# B&R Automation Studio project TD52 (part 137)

#### reactorCyclic.st
```iecst
 (*******************************************************************************
reactor		THERMOREACTOR

This code is confidential AND proprietary TO the INNIO Company.
It may NOT be used in any form, or reproduced in any manner,
without the express written permission OF the INNIO Company.
Copyright, INNIO Company, 2019

Customized modifications: -
------------------------

History:
-------
V15 	27-09-2001	Thaler, generated
V180	06-03-2003	Thaler, TR_ON_moduleTR, TR_OPER_moduleTR added. Connection to recipe REACTOR.
                            FGDRPS_moduleTR from FRG_GASREG_moduleTR --> reactor_a.
                            reactor_a --> TRW08.
V203	05-09-2003	Thaler, Modifications so that compatible with DIA.NE XT:
							y_HE_ramp INT --> UINT (reason: AS V2.3)
							Filter: 3 --> 10 (reason: AT664)
							DI_x: Value defined (reason: disabling #40 at Package Test).
							TK1, TK2 local --> global (reason: diagnosis for Development).
V210	28-09-2004	Thaler, TempInTR_moduleTR, TempOutTR_moduleTR, y_HE_Prom_moduleTR added.
							TK_GAS_OFF added.
							FG_HEIZG_moduleTR local --> global.
							TK_GAS.IN   := TK1_TK2_MIN; (war TK1_TK2_MIT).
							AN_PGW1 --> FG_TH_moduleTR.
V210.1	23-05-2006	Thaler, bExhReactor_moduleTR, Spuelluft-Ventil added.
V220    21-12-2007  Thaler, --> X20: variables declaration,
                            calculation Tvgl_moduleTR, iAT6402ETCreactor_moduleTR.
V220.2  27-05-2008  Thaler, DO_HE_xy added, TP_BTRB 180" --> DO_GAS_MINUS_moduleTR, ...
V250    12-03-2009  Thaler, UM_E_NEU_moduleTR: new position switches added.
                            TK_GAS_OFF settings changed.
V2.50.1 08-07-2009  Thaler, Spuelluft-Ventil modified.
                            Compensation_AI_TK_moduleTR added.
V3.20.0 11-03-2011  Thaler, with/without gas injection added:
                              sel_woGas: TK_w, TKx_y_HI_Gw, FRG_GASREG_moduleTR, PTON_KL_AUS
                              TK_w_woGas: TK_w
                              set_PT_KL_Pinc: PTON_KL_AUS
                              PT_KL_Pinc: PTON_KL_AUS.
                            alarm reset:
                              alarms unlatched for XT_Version_32x added
                              DI_QUITT_LT deleted (used for stand alone version only).
                            replaced variables:
                              M_GS_EIN --> DI_GCB_ON_moduleTR, NS_EIN -->  DI_MCB_ON_moduleTR
                            Spuelluft-Ventil modified:
                              TON_SPLU_AKT_AUS/EIN: 60s --> 10s
                              TON_SPLU_DEAKT: 60s --> 30s
V3.20.1 10-06-2011  Thaler, variabled deleted for simplifying Modular Software.
    	10-06-2011	Thaler, last modification
                            NOT compatible with other XT Versions !!

V04.00.00.00 	03-04-2014  Ganguly		HALio signals for 5 postion feedback and 4 postion feedback have same name,
							 			 in case of 4 position Mid-position feedback remains unconnected.
V04.03.00.00	25-09-2014	Denk		Bugfix, Flap switching time (INT/REAL casting)
										 Bugfix, KL_EIN renamed with OUT_TR.bThR_Val_SetIn
										 TRW01 : "FUEHLERBRUCH", TRW01_TempInOut and TRW01_Tvgl deleted
										 Bugfix, Sammelstoerung Reaktor Stop und Reaktor Stop + Motor Stop
V04.07.00.00	27-05-2019	Denk		Adjustments regarding new library versions (JEW_LIB1, JEW_LIB2, JEW_LIB3)
V04.09.00.00	09-03-2020	Denk		Bugfix, input variable changed in function xTON_TK1_DIF()
V04.12.00.00	19-05-2022	Maran		Bugfix: updated electrical heating elements switching logic and trigger signal for hour counter,
										 Bugfix: absolute value used for max. temperature difference detection in reactor vessel n.2,
										 Bugfix: HMI para used for aux.gas injection min. temperature hysteresis instead of fixed value,
										 removed unused TON for electrical heating thresholds detection
				14-06-2022	Maran		Removed unused TON for min.temperature detection to release auxiliary gas injection,
										 removed unused block of auxiliary gas injection release based on upper temperature bound
										 added A2356, A2357, A2358 in collective panel fault indication
V04.13.00.00	27-03-2023	Maran		Updated operating temperature definition and maximum temperature difference monitoring in TK1 and in TK2 (W3503)
				28-11-2023	Maran		Added W9374, W9375, W9376, W9377, W9381 in collective panel fault indication
V04.14.00.00	27-11-2024	Maran		Added auxiliary gas stop due to sufficient temperature,
										 temperature setpoint reference used in task changed from heating controller out structure value to HMI parameter value
				27-11-2024	Maran		Updates for thermal reactor 2nd generation (ThR2): revision of reactor chamber reference temperature,
										 added control of auxiliary gas solenoid valve before 4-way flap, adapted W3504 and blocked W3503,
										 added ThR2 chamber temperature signal fault to th.reactor bypass conditions, added ThR2 electrical heating control

Instructions for use:
--------------------

Outstandings:
------------
	FUB fuer ls und ls_t inkl. EN (ENABLE)
*******************************************************************************)
PROGRAM _CYCLIC

	xTON_INIT (IN:= TRUE, PT:= T#1m);
	OUT_TR.bThR_Active := xTON_INIT.Q AND IN_TR.tPB2MM.bParaSetupOk AND Para.bThR_Active;

	(* TK_moduleTR setpoint *)
	IF Para.bThR_woGas THEN
		TK_w := Para.rT_ThR_SetwoGas;    (* 0,1°C; without gas injection: see task "reac_set" *)
	ELSE
		TK_w := Para.tCtrTR_Heater.W_set;     (* Thermal reactor gas heating controller setpoint parameter *)
	END_IF;

	(* Temperature Limits [FB33] *)
	IF Para.bThR_woGas THEN
		TKx_y_HI_Gw       := 850.0;  (* 0,1°C; without gas injection: 850,0°C *)
	ELSE
		TKx_y_HI_Gw       := 800.0;  (* 0,1°C; with gas injection Standard: 800,0°C *)
	END_IF;

	(* Klappenumschaltzeit [FB40] *)
	(* Flap switching time *)
	PT_KL.x1 := REAL_TO_INT(TK_w + Para.rT_ThR_Val_x1);		(* von Rezept, 0,1°C; Standard: 20,0°C *)
	PT_KL.x2 := REAL_TO_INT(TK_w + Para.rT_ThR_Val_x2);		(* von Rezept, 0,1°C; Standard: 40,0°C *)
	PT_KL.y1 := TIME_TO_INT(Para.ti_ThR_Val_y1/1000);		(* von Rezept, Sekunden bei x1; Standard: 180s *)
	PT_KL.y2 := TIME_TO_INT(Para.ti_ThR_Val_y2/1000);		(* von Rezept, Sekunden bei x2; Standard: 360s *)

	(* Tvgl20_moduleTR von Rezept, 0,1°C; Standard: 0,0°C
	   Hier wird jener Wert angegeben,
	   den das Vergleichsstellenmessgeraet
	   bei 20° Umgebungstemperatur ausgibt. *)

	(******************************************************************************)
	(* Thermal Reactor temperature failure, min, max *)
	IF NOT Para.bThR2_Ena THEN //with Thermal reactor 1st generation
		MS_TK := (NOT IN_TR.tT_ThR_Chamber1_1.GoodQual) OR
				 (NOT IN_TR.tT_ThR_Chamber1_2.GoodQual) OR
				 (NOT IN_TR.tT_ThR_Chamber2_1.GoodQual) OR
				 (NOT IN_TR.tT_ThR_Chamber2_2.GoodQual);

		TK1 := (IN_TR.tT_ThR_Chamber1_1.Ai + IN_TR.tT_ThR_Chamber1_2.Ai)/2;
		TK2 := (IN_TR.tT_ThR_Chamber2_1.Ai + IN_TR.tT_ThR_Chamber2_2.Ai)/2;
	ELSE
		MS_TK := FALSE;
	END_IF
	IF Para.bThR2_Ena THEN //with Thermal reactor 2nd generation
		// individual measurement signal faults are defined with Thermal reactor 2, faults on left and right chamber are also used for reactor bypass
		bThR2_T_fault_ReactChamber := (NOT IN_TR.tThR2_T_UnitOk_RightCh.Di OR NOT IN_TR.tT_ThR2_RightChamber.GoodQual) OR
										(NOT IN_TR.tThR2_T_UnitOk_LeftCh.Di OR NOT IN_TR.tT_ThR2_LeftChamber.GoodQual);

		TK1 := IN_TR.tT_ThR2_RightChamber.Ai;
		TK2 := IN_TR.tT_ThR2_LeftChamber.Ai;
	ELSE
		bThR2_T_fault_ReactChamber := FALSE;
	END_IF

	TK1_TK2_MIT := (TK1 + TK2) / 2;
	TK1_TK2_MIN := MIN (TK1, TK2);
	TK1_TK2_MAX := MAX (TK1, TK2);
	(******************************************************************************)

	(* Steuerprogramm (aus PB4) *)

	(* Freigabe Thermoreaktor von Modulsteuerung *)
	(* Release Thermal Reactor from Module controller *)
	xTON_FG_TH (IN:= ((bThR_Rel AND IN_TR.tGCB_On.Di AND IN_TR.tMCB_On.Di) OR bThR_RelTest), PT:= T#30s);

	(* Freigabe Abgasklappen-Umschaltung und el. Heizung *)
	FG_KLUM						:= OUT_TR.bThR_Active AND xTON_FG_TH.Q AND
								    IN_TR.tThR_Swth_On.Di AND NOT ST_R_ST AND NOT ST_RM_ST;
	FG_HEIZG_moduleTR			:= FG_KLUM;
	OUT_TR.tThR_Contactor.Do	:= FG_HEIZG_moduleTR;
	OUT_TR.bThR_RelHeat			:= FG_HEIZG_moduleTR;

	(* Thermal Reactor auxiliary gas stop due to sufficient temperature *)
	bThr_AuxGasStopT_Ena := NOT Para.bThR_woGas AND Para.bThR_auxGasMonitor AND Para.bCtrThR_Heater_Active AND (TK_w > Para.rT_ThR_LimGas); (* check on parameters consistency *)

	xTON_Thr_AuxGasStopT_set(IN := OUT_TR.bThR_RelGas AND (IN_TR.tPos_ThR_AuxGasCV_Act.Ai < rPos_ThR_GasCV_AuxGasStop_max) (*CV essentially closed *) AND
	 IN_TR.tPos_ThR_AuxGasCV_Act.GoodQual AND (TK_moduleTR > TK_w + rT_Thr_AuxGasStopT_rel), PT := tiTON_Thr_AuxGasStopT_set);
	xRS_Thr_AuxGasStopT.SET := xTON_Thr_AuxGasStopT_set.Q; (* activation *)

	xTON_Thr_AuxGasStopT_reset(IN := (TK_moduleTR < TK_w), PT := tiTON_Thr_AuxGasStopT_reset);
	xRS_Thr_AuxGasStopT.RESET1 := xTON_Thr_AuxGasStopT_reset.Q OR NOT FG_HEIZG_moduleTR OR NOT bThr_AuxGasStopT_Ena; (* deactivation *)

	xRS_Thr_AuxGasStopT();

	(* Freigabe Einduesung *)
	OUT_TR.bThR_RelGas     := FG_HEIZG_moduleTR AND xTK_GAS.QH AND NOT Para.bThR_woGas AND NOT xRS_Thr_AuxGasStopT.Q1;
	OUT_TR.tThR_GT_COn1.Do := OUT_TR.bThR_RelGas;
	OUT_TR.tThR_GT_COn2.Do := OUT_TR.bThR_RelGas;
	OUT_TR.bThR_RelGas_Tmin	:= xTK_GAS.QH; (* minimum temperature for gas injection reached *)

	(* Betriebsmeldung *)
	OUT_TR.tThR_RunLamp.Do := (FG_KLUM AND (SEK_TAKT OR xTK_OPER.QH)) OR IN_TR.tThR_LampTest.Di;

	(* Betriebsmeldungen fuer auftragsbezogene Verwendung *)
	OUT_TR.bThR_Run         := FG_KLUM;               	    (* Reaktor eingeschaltet *)
	OUT_TR.bThR_RunReacTemp := FG_KLUM AND xTK_OPER.QH;	(* Reaktor eingeschaltet, Reaktionstemp. erreicht *)

	(* Ansteuerung Spuelluft-Stopp-Ventil, neu hinzu 07-2009 *)
	(* Aktivierung Spuelluft vor Durchfuehrung der Klappenbewegung *)
	PTON_SPLU_AKT_AUS := LIMIT (0, PTON_KL_AUS - T#10s, PTON_KL_AUS);
	PTON_SPLU_AKT_EIN := LIMIT (0, PTON_KL_EIN - T#10s, PTON_KL_EIN);
	xTON_SPLU_AKT_AUS (IN:= OUT_TR.bThR_Val_SetOut, PT:= PTON_SPLU_AKT_AUS);
	xTON_SPLU_AKT_EIN (IN:= OUT_TR.bThR_Val_SetIn, PT:= PTON_SPLU_AKT_EIN);

	(* Ansteuerung Spuelluft-Stopp-Ventil, neu hinzu 05-2006, modifiziert 07-2009 *)
	(* Deaktivierung Spuelluft nach Durchfuehrung der Klappenbewegung *)
	xTON_SPLU_DEAKT (IN:= (NOT FG_KLUM OR RM_KL_END), PT := T#30s);

	IF xTON_SPLU_DEAKT.Q THEN
		SPLU_AKT := FALSE;
	END_IF;

	(* IF FG_KLUM AND NOT OUT_TR.b_ThR_Val_SetIn AND NOT OUT_TR.b_ThR_Val_SetOut THEN *)
	IF (FG_KLUM AND NOT RM_KL_END) OR
	   (FG_KLUM AND (xTON_SPLU_AKT_AUS.Q OR xTON_SPLU_AKT_EIN.Q)) THEN
		SPLU_AKT := TRUE;
	END_IF;

	xTOF_W_INT (IN:= (IN_TR.tThR_Swth_On.Di AND xTON_W_ACT.Q), PT := T#10050m);	  (* weekly SPLU interval *)
	xTON_W_ACT (IN:= (IN_TR.tThR_Swth_On.Di AND NOT xTOF_W_INT.Q), PT := T#30m);  (* weekly SPLU active *)

	OUT_TR.tThR_Val_Air.Do := NOT (SPLU_AKT OR (IN_TR.tThR_Swth_On.Di AND NOT xTOF_W_INT.Q));	(* Ausgang fuer Spuelluft-Stopp-Ventil, TRUE bei STOP *)

	(* Klappensteuerung (aus OB13, FB35, FB36) *)

	(* Abgasklappe Mittelstellung: *)
	(* Im spannungslosen Zustand der Ansteuerventile geht die Klappe auf Mittelstellung. *)
	IF NOT FG_KLUM AND NOT Para.bSel_FlapActEl THEN
		OUT_TR.tThR_Val_CCylIn.Do  := FALSE;
		OUT_TR.tThR_Val_CCylOut.Do := FALSE;
	END_IF;

	(* Klappe Mittelstellung erreicht *)
	RM_KL_MIT :=          IN_TR.tPos_ThR_Val_Mid.Di
	              AND NOT IN_TR.tPos_ThR_Val_In1.Di
		          AND NOT IN_TR.tPos_ThR_Val_In2.Di
		          AND NOT IN_TR.tPos_ThR_Val_Out1.Di
				  AND NOT IN_TR.tPos_ThR_Val_Out2.Di;

	(* Abgasklappe Umschaltung: *)
	IF FG_KLUM THEN
		xR_TRIG_KL_AUS (CLK:= OUT_TR.bThR_Val_SetOut);
		xR_TRIG_KL_EIN (CLK:= OUT_TR.bThR_Val_SetIn);

		(* Bei positiver Flanke von KL_EIN_moduleTR oder KL_AUS_moduleTR sowie wenn KL_EIN_moduleTR und KL_AUS_moduleTR
		   nicht anstehen, wird die Mittelstellung aktiviert. *)
		IF (xR_TRIG_KL_AUS.Q OR xR_TRIG_KL_EIN.Q OR (OUT_TR.bThR_Val_SetOut AND OUT_TR.bThR_Val_SetIn)) THEN
			OUT_TR.tThR_Val_CCylIn.Do  := FALSE;
			OUT_TR.tThR_Val_CCylOut.Do := FALSE;
		END_IF;

		(* Klappe Ausfahren:
		   - Anfahren Mittelstellung durch Y1=0, Y2=0
		   - Rueckmeldung Mittelstellung erreicht: Ausfahren durch Aktivieren von Y2
		   - Ueberwachung:
		     Falls nach 10" die Endlage nicht erreicht wird,
		       "Stoerung Abgasklappe Ende" mit Reaktorabschaltung und
		       Befehl Abgasklappe Mittelstellung.
		     Falls 5" danach die Mittelstellung nicht erreicht wird,
		       "Stoerung Abgasklappe Mittelstellung" mit Gasmotorabstellung. *)
		IF OUT_TR.bThR_Val_SetOut THEN
			OUT_TR.tThR_Val_CCylIn.Do := FALSE;
		END_IF;

		IF (OUT_TR.bThR_Val_SetOut AND RM_KL_MIT) THEN
			OUT_TR.tThR_Val_CCylOut.Do := TRUE;
		END_IF;

		(* Klappe Einfahren:
		   - Anfahren Mittelstellung durch Y1=0, Y2=0
	   	   - Rueckmeldung Mittelstellung erreicht: Einfahren durch Aktivieren von Y1
		   - Ueberwachung:
		     Falls nach 10" die Endlage nicht erreicht wird,
		       "Stoerung Abgasklappe Ende" mit Reaktorabschaltung und
		       Befehl Abgasklappe Mittelstellung.
		     Falls 5" danach die Mittelstellung nicht erreicht wird,
		       "Stoerung Abgasklappe Mittelstellung" mit Gasmotorabstellung. *)
		IF OUT_TR.bThR_Val_SetIn THEN
			OUT_TR.tThR_Val_CCylOut.Do := FALSE;
		END_IF;

		IF (OUT_TR.bThR_Val_SetIn AND RM_KL_MIT) THEN
			OUT_TR.tThR_Val_CCylIn.Do := TRUE;
		END_IF;
	END_IF;

	(* Klappe Endlage erreicht *)
	RM_KL_END     := (	OUT_TR.bThR_Val_SetOut
					AND IN_TR.tPos_ThR_Val_Out1.Di
					AND IN_TR.tPos_ThR_Val_Out2.Di
					AND NOT IN_TR.tPos_ThR_Val_In1.Di
					AND NOT IN_TR.tPos_ThR_Val_In2.Di
					AND NOT IN_TR.tPos_ThR_Val_Mid.Di)
				  OR
					(	OUT_TR.bThR_Val_SetIn
					AND IN_TR.tPos_ThR_Val_In1.Di
					AND IN_TR.tPos_ThR_Val_In2.Di
					AND NOT IN_TR.tPos_ThR_Val_Out1.Di
					AND NOT IN_TR.tPos_ThR_Val_Out2.Di
					AND NOT IN_TR.tPos_ThR_Val_Mid.Di);

	RM_KL_END_AUS := (  IN_TR.tPos_ThR_Val_Out1.Di
					AND IN_TR.tPos_ThR_Val_Out2.Di
					AND NOT IN_TR.tPos_ThR_Val_In1.Di
					AND NOT IN_TR.tPos_ThR_Val_In2.Di
					AND NOT IN_TR.tPos_ThR_Val_Mid.Di);

	RM_KL_END_EIN := (  IN_TR.tPos_ThR_Val_In1.Di
					AND IN_TR.tPos_ThR_Val_In2.Di
					AND NOT IN_TR.tPos_ThR_Val_Out1.Di
					AND NOT IN_TR.tPos_ThR_Val_Out2.Di
					AND NOT IN_TR.tPos_ThR_Val_Mid.Di);

	(* Abgasklappe Einschaltung Schütze mit E-Antrieb: *)
	(* Abgasklappe Mittelstellung mit E-Antrieb: *)
	IF NOT FG_KLUM AND Para.bSel_FlapActEl THEN
		R_TRIG_KL_AUS_M (CLK:= KL_AUS_M);
		R_TRIG_KL_EIN_M (CLK:= KL_EIN_M);
		OUT_TR.tThR_Val_CCylOut.Do := R_TRIG_KL_AUS_M.Q;
		OUT_TR.tThR_Val_CCylIn.Do  := R_TRIG_KL_EIN_M.Q;
	END_IF;
	(* Anmerkung: Selbsthaltung extern mit Schütz, Absteuerung mit Endschalter Mittelstellung *)

	(* Abgasklappe Umschaltung mit E-Antrieb: *)
	IF FG_KLUM AND Para.bSel_FlapActEl THEN

		(* Klappe Ausfahren:
	   	   - Rueckmeldung Endlage_Eingefahren oder Mittelstellung erreicht:
	         Ausfahren durch Dauerbefehl *)

		(* Dauerbefehl fuer Richtungswechsel *)
		IF (OUT_TR.bThR_Val_SetOut AND (RM_KL_MIT OR RM_KL_END_EIN)) THEN
			OUT_TR.tThR_Val_CCylOut.Do := TRUE;
		END_IF;

		(* Klappe Einfahren:
	   	   - Rueckmeldung Endlage_Ausgefahren oder Mittelstellung erreicht:
	         Einfahren durch Dauerbefehl *)

		(* Dauerbefehl fuer Richtungswechsel *)
		IF (OUT_TR.bThR_Val_SetIn AND (RM_KL_MIT OR RM_KL_END_AUS)) THEN
			OUT_TR.tThR_Val_CCylIn.Do := TRUE;
		END_IF;
	END_IF;

	(* Zeittakte Abgasklappe Umschaltung *)
	OUT_TR.bThR_Val_SetOut  := FG_KLUM
							AND (NOT xTON_KL_AUS.Q)
							AND (NOT OUT_TR.bThR_Val_SetIn)
							AND (OUT_TR.bThR_Val_SetOut OR NOT KL_AUS_S);

	IF OUT_TR.bThR_Val_SetOut THEN
		KL_AUS_S   := TRUE;
		KL_AUS_M_S := TRUE;
		KL_EIN_S   := FALSE;
		KL_EIN_M_S := FALSE;
	END_IF;
	xTON_KL_AUS (IN:= OUT_TR.bThR_Val_SetOut, PT:= PTON_KL_AUS);

	OUT_TR.bThR_Val_SetIn := FG_KLUM
						AND (NOT xTON_KL_EIN.Q)
						AND (NOT OUT_TR.bThR_Val_SetOut)
						AND TRUE;

	IF OUT_TR.bThR_Val_SetIn THEN
		KL_EIN_S   := TRUE;
		KL_EIN_M_S := TRUE;
		KL_AUS_S   := FALSE;
		KL_AUS_M_S := FALSE;
	END_IF;
	xTON_KL_EIN (IN:= OUT_TR.bThR_Val_SetIn, PT:= PTON_KL_EIN);

	(* Abgasklappe Mittelstellung mit E-Antrieb: *)
	(* Zeittakte Abgasklappe für Anfahren Mittelstellung mit E-Antrieb: *)
	xTOF_S_EIN (IN:= (Para.bThR_Active AND IN_TR.tThR_Swth_On.Di), PT:= T#15s);
	xTON_FG_KL_M (IN:= (xTOF_S_EIN.Q AND NOT FG_KLUM AND NOT RM_KL_MIT AND NOT xTRA01M.Q1), PT:= T#1s);
	FG_KL_M := xTON_FG_KL_M.Q;

	KL_AUS_M := FG_KL_M AND NOT xTON_KL_AUS_M.Q AND NOT KL_EIN_M AND
				(KL_AUS_M OR NOT KL_AUS_M_S OR RM_KL_END_EIN);
	IF KL_AUS_M THEN
		KL_AUS_M_S := TRUE;
		KL_EIN_M_S := FALSE;
	END_IF;
	xTON_KL_AUS_M (IN:= KL_AUS_M, PT:= T#5s);

	KL_EIN_M := FG_KL_M AND NOT xTON_KL_EIN_M.Q AND NOT KL_AUS_M AND TRUE;
	IF KL_EIN_M THEN
		KL_EIN_M_S := TRUE;
		KL_AUS_M_S := FALSE;
	END_IF;
	xTON_KL_EIN_M (IN:= KL_EIN_M, PT:= T#5s);

	(* Abgasklappe Umschaltung mit E-Antrieb: *)
	IF FG_KLUM AND Para.bSel_FlapActEl THEN

		(* Klappe Ausfahren:
	       - Rueckmeldung Endlage_Eingefahren oder Mittelstellung erreicht:
	         Ausfahren durch Dauerbefehl (siehe oberhalb)
	       - Rueckmeldung Endlage_Ausgefahren: Beendigung Dauerbefehl
	       - Ueberwachung:
	         Falls nach 10" die Endlage nicht erreicht wird,
	         "Stoerung Abgasklappe Ende" mit Reaktorabschaltung und
	         Befehl Abgasklappe Mittelstellung.
	         Falls 5" danach die Mittelstellung nicht erreicht wird,
	         "Stoerung Abgasklappe Mittelstellung" mit Gasmotorabstellung. *)

		(* Absteuerung *)
		IF (OUT_TR.bThR_Val_SetOut AND RM_KL_END_AUS) OR NOT OUT_TR.bThR_Val_SetOut THEN
			OUT_TR.tThR_Val_CCylOut.Do := FALSE;
		END_IF;

		(* Klappe Einfahren:
	   	   - Rueckmeldung Endlage_Ausgefahren oder Mittelstellung erreicht:
	      	 Einfahren durch Dauerbefehl (siehe oberhalb)
	   	   - Rueckmeldung Endlage_Eingefahren: Beendigung Dauerbefehl
	   	   - Ueberwachung:
	     	 Falls nach 10" die Endlage nicht erreicht wird,
	       	 "Stoerung Abgasklappe Ende" mit Reaktorabschaltung und
	       	 Befehl Abgasklappe Mittelstellung.
	     	 Falls 5" danach die Mittelstellung nicht erreicht wird,
	       	 "Stoerung Abgasklappe Mittelstellung" mit Gasmotorabstellung. *)

		(* Absteuerung *)
		IF (OUT_TR.bThR_Val_SetIn AND RM_KL_END_EIN) OR NOT OUT_TR.bThR_Val_SetIn THEN
			OUT_TR.tThR_Val_CCylIn.Do  := FALSE;
		END_IF;
	END_IF;

	(* Abgasklappe Verriegelung mit E-Antrieb: *)
	IF Para.bSel_FlapActEl THEN
		IF OUT_TR.bThR_Val_SetOut OR KL_AUS_M THEN
			OUT_TR.tThR_Val_CCylIn.Do  := FALSE;
		END_IF;
		IF OUT_TR.bThR_Val_SetIn OR KL_EIN_M THEN
			OUT_TR.tThR_Val_CCylOut.Do  := FALSE;
		END_IF;
	END_IF;

	(* Abgasklappe Mittelstellung mit Druckluft-Anztrieb: *)
	(* Im spannungslosen Zustand der Ansteuerventile geht die Klappe auf Mittelstellung. *)
	IF NOT FG_KLUM AND NOT Para.bSel_FlapActEl THEN
		OUT_TR.tThR_Val_CCylIn.Do  := FALSE;
		OUT_TR.tThR_Val_CCylOut.Do := FALSE;
	END_IF;

	(* Abgasklappe Umschaltung mit Druckluft-Antrieb: *)
	IF FG_KLUM AND NOT Para.bSel_FlapActEl THEN
		R_TRIG_KL_AUS (CLK:= OUT_TR.bThR_Val_SetOut);
		R_TRIG_KL_EIN (CLK:= OUT_TR.bThR_Val_SetIn);

		(* Bei positiver Flanke von KL_EIN oder KL_AUS sowie wenn KL_EIN und KL_AUS
	    nicht anstehen, wird die Mittelstellung aktiviert. *)
		IF (R_TRIG_KL_AUS.Q OR R_TRIG_KL_EIN.Q OR (OUT_TR.bThR_Val_SetOut AND OUT_TR.bThR_Val_SetIn)) THEN
			OUT_TR.tThR_Val_CCylIn.Do  := FALSE;
			OUT_TR.tThR_Val_CCylOut.Do := FALSE;
		END_IF;

		(* Klappe Ausfahren:
	       - Anfahren Mittelstellung durch Y1=0, Y2=0
	       - Rueckmeldung Mittelstellung erreicht: Ausfahren durch Aktivieren von Y2
	       - Ueberwachung:
	       Falls nach 10" die Endlage nicht erreicht wird,
	       "Stoerung Abgasklappe Ende" mit Reaktorabschaltung und
	       Befehl Abgasklappe Mittelstellung.
	       Falls 5" danach die Mittelstellung nicht erreicht wird,
	       "Stoerung Abgasklappe Mittelstellung" mit Gasmotorabstellung. *)
		IF OUT_TR.bThR_Val_SetOut THEN
			OUT_TR.tThR_Val_CCylIn.Do := FALSE;
		END_IF;
		IF (OUT_TR.bThR_Val_SetOut AND RM_KL_MIT) THEN
			OUT_TR.tThR_Val_CCylOut.Do := TRUE;
		END_IF;

		(* Klappe Einfahren:
	   	   - Anfahren Mittelstellung durch Y1=0, Y2=0
	  	   - Rueckmeldung Mittelstellung erreicht: Einfahren durch Aktivieren von Y1
	       - Ueberwachung:
	     		Falls nach 10" die Endlage nicht erreicht wird,
	       		"Stoerung Abgasklappe Ende" mit Reaktorabschaltung und
	            Befehl Abgasklappe Mittelstellung.
	     		Falls 5" danach die Mittelstellung nicht erreicht wird,
	       		"Stoerung Abgasklappe Mittelstellung" mit Gasmotorabstellung. *)
		IF OUT_TR.bThR_Val_SetIn THEN
			OUT_TR.tThR_Val_CCylOut.Do := FALSE;
		END_IF;
		IF (OUT_TR.bThR_Val_SetIn AND RM_KL_MIT) THEN
			OUT_TR.tThR_Val_CCylIn.Do := TRUE;
		END_IF;
	END_IF;

	(* Thermal Reactor auxiliary gas solenoid valve - ThR2 *)
	IF Para.bThR2_Ena THEN
		IF OUT_TR.bThR_RelGas THEN
			//update blockage function inputs before 4-way flap switching request depending on last end-position
			IF iThr2_lastFlapEndPosIndex = 1 THEN
				xSR_Thr2_AuxGasValve_Block.SET1 := xTON_KL_EIN.PT - xTON_KL_EIN.ET <= tiThR2_AuxGasValve_Block;
				xSR_Thr2_AuxGasValve_Block.RESET := RM_KL_END_AUS;
			ELSIF iThr2_lastFlapEndPosIndex = -1 THEN
				xSR_Thr2_AuxGasValve_Block.SET1 := xTON_KL_AUS.PT - xTON_KL_AUS.ET <= tiThR2_AuxGasValve_Block;
				xSR_Thr2_AuxGasValve_Block.RESET := RM_KL_END_EIN;
			END_IF
		ELSE //reinitialize blockage function inputs in case of Th.Reactor aux.gas system stop
			xSR_Thr2_AuxGasValve_Block.SET1 := FALSE;
			xSR_Thr2_AuxGasValve_Block.RESET := TRUE;
		END_IF
		xSR_Thr2_AuxGasValve_Block();
		OUT_TR.tThR2_AuxGasShutOffValve_Dem.Do := OUT_TR.bThR_RelGas AND RM_KL_END AND (NOT xSR_Thr2_AuxGasValve_Block.Q1);
	ELSE
		//reset SR in IF block
		xSR_Thr2_AuxGasValve_Block.SET1 := FALSE;
		xSR_Thr2_AuxGasValve_Block.RESET := TRUE;
		//reset output signal gas solenoid valve - ThR2
		OUT_TR.tThR2_AuxGasShutOffValve_Dem.Do := FALSE;
	END_IF
	IF OUT_TR.bThR_RelGas THEN //record last end-position reached by 4-way flap during aux. gas. injection operation
		IF RM_KL_END_EIN THEN
			iThr2_lastFlapEndPosIndex := 1; //right position
		ELSIF RM_KL_END_AUS THEN
			iThr2_lastFlapEndPosIndex := -1; //left position
		END_IF
	ELSE
		iThr2_lastFlapEndPosIndex := 0; //reset position index
	END_IF

	//block the auxiliary gas heating controller if corresponding solenoid valve is closed
	bThr2_AuxGasValve_CtrlBlock := Para.bThR2_Ena AND OUT_TR.bThR_RelGas AND NOT OUT_TR.tThR2_AuxGasShutOffValve_Dem.Do;

	(******************************************************************************)
	(******************************************************************************)

	(* Ueberwachungen [PB45] *)

	(* TRA01 : "STOERUNG ABGASKLAPPE MITTELSTELLUNG" *)
	xTON_ST_KLM.IN := OUT_TR.bThR_Active AND NOT FG_KLUM AND NOT RM_KL_MIT AND NOT xTON_ST_KLM.Q AND NOT xTRA01M.RESET;
	xTON_ST_KLM.PT := T#15s;
	xTON_ST_KLM;
	xTRA01.SET1  := xTON_ST_KLM.Q;
	xTRA01.RESET := NOT xTRA01.SET1;
	xTRA01();
	xTRA01M.SET1  := xTON_ST_KLM.Q;
	xTRA01M.RESET := IN_TR.tAB2TR.bResetTrip;
	xTRA01M();

	(* TRA02 : "SICHERHEITSSCHLEIFE THERMOREAKTOR", aktiv nur bei RIO *)
	xTRA02.SET1  := IN_TR.tThR_SL.Di;
	xTRA02.RESET := NOT xTRA02.SET1;
	xTRA02();

	(* TRW01 : "FUEHLERBRUCH" *)
	xTRW01_TK.SET1  := MS_TK;
	xTRW01_TK.RESET := NOT xTRW01_TK.SET1;
	xTRW01_TK();
	xTRW01.SET1  := xTRW01_TK.Q1;
	xTRW01.RESET := NOT xTRW01.SET1;
	xTRW01();

	(* TRW02 : "STOERUNG DRUCKLUFTVERSORGUNG" *)
	xTOF_PS_LUFT (IN:= IN_TR.tPr_ThR_AirLo.Di  AND NOT Para.bSel_FlapActEl, PT := T#10s);
	xTRW02.SET1  := Para.bThR_Active AND NOT xTOF_PS_LUFT.Q AND NOT Para.bSel_FlapActEl;
	xTRW02.RESET := NOT xTRW02.SET1;
	xTRW02();

	(* TRW03 : "STOERUNG ABGASKLAPPE ENDLAGE" *)
	xTON_ST_KLE (IN:= ((OUT_TR.bThR_Val_SetOut AND NOT RM_KL_END_AUS) OR
					   (OUT_TR.bThR_Val_SetIn  AND NOT RM_KL_END_EIN)), PT:= T#10s);
	xTRW03.SET1  := xTON_ST_KLE.Q;
	xTRW03.RESET := NOT xTRW03.SET1;
	xTRW03();

	(* TRW04 : "AUFHEIZZEIT UEBERSCHRITTEN" *)
	xTON_AUFHEIZG_GES (IN:= (FG_KLUM AND NOT xTK_OPER.QH), PT:= T#600m);
	xTON_AUFHEIZG_GAS (IN:= (OUT_TR.bThR_RelGas AND NOT xTK_OPER.QH), PT:= T#300m);
	xTRW04.SET1  := xTON_AUFHEIZG_GES.Q OR xTON_AUFHEIZG_GAS.Q;
	xTRW04.RESET := NOT xTRW04.SET1;
	xTRW04();

	(* TRW05 : "SCHALTSCHRANKTEMPERATUR MAXIMUM" *)
	xTRW05.SET1  := OUT_TR.bThR_Active AND NOT IN_TR.tT_ThR_Swg_Hi.Di;
	xTRW05.RESET := NOT xTRW05.SET1;
	xTRW05();

	(* TRW06 : "ZULAESSIGE DIFFERENZ VON TEMPERATUREN TK1/TK2 UEBER MAXIMUM" *)
	xTRW06.SET1  := xTK1_DIF_HI.QH OR xTK2_DIF_HI.QH;
	xTRW06.RESET := NOT xTRW06.SET1;
	xTRW06();

	(* TRW07 : "TEMPERATUR REAKTIONSKAMMER TK1/TK2 MAXIMUM" *)
	IF NOT Para.bThR2_Ena THEN //with Thermal reactor 1st generation
		xTRW07.SET1  := xTK1_1_HI.QH OR xTK1_2_HI.QH OR xTK2_1_HI.QH OR xTK2_2_HI.QH;
	END_IF
	IF Para.bThR2_Ena THEN //with Thermal reactor 2nd generation
	   (*************** temperature threshold check for TRW07 - ThR2 ***************)
		xGRMax_ThR2_T_LeftChamber_Hi(Gw := TKx_y_HI_Gw, Hy := TKx_y_HI_Hy, In := IN_TR.tT_ThR2_LeftChamber.Ai);
		xTON_ThR2_T_LeftChamber_Hi(IN := xGRMax_ThR2_T_LeftChamber_Hi.Q, PT := ti_TKx_y_HI_PTHI);

		xGRMax_ThR2_T_RightChamber_Hi(Gw := TKx_y_HI_Gw, Hy := TKx_y_HI_Hy, In := IN_TR.tT_ThR2_RightChamber.Ai);
		xTON_ThR2_T_RightChamber_Hi(IN := xGRMax_ThR2_T_RightChamber_Hi.Q, PT := ti_TKx_y_HI_PTHI);

		xTRW07.SET1  := xTON_ThR2_T_LeftChamber_Hi.Q OR xTON_ThR2_T_RightChamber_Hi.Q;
	ELSE //reset TON in IF block
		xTON_ThR2_T_LeftChamber_Hi(IN := FALSE, PT := ti_TKx_y_HI_PTHI);
		xTON_ThR2_T_RightChamber_Hi(IN := FALSE, PT := ti_TKx_y_HI_PTHI);
	END_IF
	xTRW07.RESET := NOT xTRW07.SET1;
	xTRW07();

	(* TRW08 : "TEMPERATUR REAKTIONSKAMMER MINIMUM" *)
	xTRW08.SET1  := OUT_TR.bThR_Active AND NOT IN_TR.tT_ThR_ChamberLo.Di;
	xTRW08.RESET := NOT xTRW08.SET1;
	xTRW08();

	(* Sammelstoerung Reaktor Stop *)
	IF IN_TR.tAB2TR.bResetWarning THEN
		ST_R_ST := FALSE;
	END_IF;

	IF (xTRW01_TK.Q1
		OR bThR2_T_fault_ReactChamber
		OR xTRW02.Q1
		OR xTRW03.Q1
		OR xTRW04.Q1
		OR xTRW05.Q1
		OR xTRW06.Q1
		OR xTRW07.Q1
		OR xTRW08.Q1) THEN
		ST_R_ST := TRUE;
	END_IF;

	(* Sammelstoerung Reaktor + Motor Stop *)
	IF IN_TR.tAB2TR.bResetTrip THEN
		ST_RM_ST := FALSE;
	END_IF;

	IF FALSE (* priority 3 alarms from Th.Reactor to be included here *) THEN
		 ST_RM_ST := TRUE;
	END_IF;

	(* H2: "Reaktor Sammelstoerung", aktiv nur bei RIO *)
	OUT_TR.tThR_ErrLamp.Do
		:= xTRA01.Q1
		OR xTRA02.Q1
		OR MM2VIS.bMsg2356
		OR MM2VIS.bMsg2357
		OR MM2VIS.bMsg2358
		OR xTRW01.Q1
		OR bThR2_T_fault_ReactChamber
		OR xTRW02.Q1
		OR xTRW03.Q1
		OR xTRW04.Q1
		OR xTRW05.Q1
		OR xTRW06.Q1
		OR xTRW07.Q1
		OR xTRW08.Q1
		OR MM2VIS.bMsg9374
		OR MM2VIS.bMsg9375
		OR MM2VIS.bMsg9376
		OR MM2VIS.bMsg9377
		OR MM2VIS.bMsg9381
		OR IN_TR.tThR_LampTest.Di;

	(******************************************************************************)
	(* Auswahl der Reaktionstemperatur in Abhaengigkeit der Stroemungsrichtung [FB66] *)
	TK_moduleTR := TK1_TK2_MAX;

	(* Sekundentakt [FB3]
	CTU_SEK_TAKT (CU := FALSE, RESET := CTU_SEK_TAKT.Q, PV := 10);
	CTU_SEK_TAKT (CU := TRUE, RESET := CTU_SEK_TAKT.Q, PV := 10);
	SEK_TAKT := (CTU_SEK_TAKT.CV >= 5) AND (CTU_SEK_TAKT.CV <= 10);
	*)

	xTON_reactor_01.IN := NOT(SEK_TAKT);
	xTON_reactor_01.PT := T#300ms;
	xTON_reactor_01();

	IF (xTON_reactor_01.Q = 1) THEN
		SEK_TAKT := 1;
	END_IF;

	xTON_reactor_02.IN := SEK_TAKT;
	xTON_reactor_02.PT := T#600ms;
	xTON_reactor_02();

	IF (xTON_reactor_02.Q = 1) THEN
		SEK_TAKT := 0;
	END_IF;

	IF NOT Para.bThR2_Ena THEN // El. heating with Thermal reactor 1st generation
		(* Heizstabsteuerung [FB45, FB56]
		   Periodendauer = 4*100ms.
		   Impulsdauer   = 0...4*100ms. *)
		xCTD_HE_1 (CD := FALSE, LOAD := xCTD_HE_1.Q, PV := 4);
		xCTD_HE_1 (CD := TRUE, LOAD := xCTD_HE_1.Q, PV := 4);

		(* Phasenverschiebung 2*100ms *)
		xCTD_HE_2 (CD := FALSE, LOAD := xCTD_HE_1.CV = 1, PV := 4);
		xCTD_HE_2 (CD := TRUE, LOAD := FALSE, PV := 4);

		(* Phasenverschiebung 3*100ms *)
		xCTD_HE_3 (CD := FALSE, LOAD := xCTD_HE_1.CV = 0, PV := 4);
		xCTD_HE_3 (CD := TRUE, LOAD := FALSE, PV := 4);

		IF FG_HEIZG_moduleTR = FALSE OR xTK_E00.QH THEN
			y_HE := 0;
		ELSIF FG_HEIZG_moduleTR AND NOT(xTK_E00.QH) AND xTK_E25.QH THEN
			y_HE := 1;
		ELSIF FG_HEIZG_moduleTR AND NOT(xTK_E00.QH) AND NOT(xTK_E25.QH) AND xTK_E50.QH THEN
			y_HE := 2;
		ELSIF FG_HEIZG_moduleTR AND NOT(xTK_E00.QH) AND NOT(xTK_E25.QH) AND NOT(xTK_E50.QH) AND xTK_E75.QH THEN
			y_HE := 3;
		ELSIF FG_HEIZG_moduleTR AND NOT(xTK_E00.QH) AND NOT(xTK_E25.QH) AND NOT(xTK_E50.QH) AND NOT(xTK_E75.QH) THEN
			y_HE := 4;
		ELSE
			y_HE := 0;
		END_IF;

		(* RAMP FUNCTION *)
		P_ramp[0].In         := REAL_TO_INT(y_HE * 1000);      (* "PV_In": use "PV Name" of "In" *)
		P_ramp[0].In_ref     := 1;                (* reference value, units like "In" *)
		P_ramp[0].mode       := 0;                (* 1: dOut=Ki*(In-Out)/In_ref, 0: dOut=Ki *)
		P_ramp[0].Ki_plus    := 333;              (* 0,1 units "In"/s *)
		P_ramp[0].Ki_minus   := 10000;            (* 0,1 units "In"/s *)
		P_ramp[0].dOut_max_p := 10000;            (* 0,1 units "In"/s *)
		P_ramp[0].dOut_max_m := 10000;            (* 0,1 units "In"/s *)
		P_ramp[0].Out_min    := 0;                (* units like "In" *)
		P_ramp[0].Out_max    := P_ramp[0].In;     (* units like "In" *)
		y_HE_ramp := REAL_TO_UINT(P_ramp[0].Out) / 1000;	(* "PV_Out": use "PV Name" of "Out", units like "In" *)

		rThR_EH_pulse := LIMIT(0, UINT_TO_REAL(y_HE_ramp * 100) - 10, 290);	// limit pulse duration from 0% to 75% of time interval
		tThR_EH_pulse:= REAL_TO_TIME(rThR_EH_pulse);
		xTP_EH11(IN := xCTD_HE_1.Q, PT:= tThR_EH_pulse);
		xTP_EH21(IN := xCTD_HE_2.Q, PT:= tThR_EH_pulse);
		xTP_EH31(IN := xCTD_HE_3.Q, PT:= tThR_EH_pulse);
		OUT_TR.tThR_EH11.Do := xTP_EH11.Q;
		OUT_TR.tThR_EH21.Do := xTP_EH21.Q;
		OUT_TR.tThR_EH31.Do := xTP_EH31.Q;
		IF y_HE_ramp = 4 THEN 												// overwrite pulse signal for 100% heating output request
			OUT_TR.tThR_EH11.Do := OUT_TR.tThR_EH21.Do := OUT_TR.tThR_EH31.Do := 1;
		END_IF
		IF y_HE_ramp = 0 THEN 												// overwrite pulse signal for no heating output request
			OUT_TR.tThR_EH11.Do := OUT_TR.tThR_EH21.Do := OUT_TR.tThR_EH31.Do := 0;
		END_IF

		OUT_TR.tThR_EH12.Do := OUT_TR.tThR_EH11.Do;
		OUT_TR.tThR_EH13.Do := OUT_TR.tThR_EH11.Do;

		OUT_TR.tThR_EH22.Do := OUT_TR.tThR_EH21.Do;
		OUT_TR.tThR_EH23.Do := OUT_TR.tThR_EH21.Do;

		OUT_TR.tThR_EH32.Do := OUT_TR.tThR_EH31.Do;
		OUT_TR.tThR_EH33.Do := OUT_TR.tThR_EH31.Do;

		IF FG_HEIZG_moduleTR THEN
			CASE y_HE_ramp OF
				0: OUT_TR.rP_ThR_EH := 0;
				1: OUT_TR.rP_ThR_EH := 250;
				2: OUT_TR.rP_ThR_EH := 500;
				3: OUT_TR.rP_ThR_EH := 750;
				4: OUT_TR.rP_ThR_EH := 1000;
			ELSE
				OUT_TR.rP_ThR_EH := 0;
			END_CASE;
		ELSE
			OUT_TR.rP_ThR_EH := 0;
		END_IF;

	ELSE
		//reset ramps/timer blocks in IF block
		P_ramp[0].Out_internal := 0;
		P_ramp[1].Out_internal := 0; //P_ramp[1] never used, reinitialized for completeness
		xTP_EH11(IN := FALSE);
		xTP_EH21(IN := FALSE);
		xTP_EH31(IN := FALSE);
	END_IF
	IF Para.bThR2_Ena THEN // El. heating with Thermal reactor 2nd generation
		//definition of five el.heating power levels
		xGRMax_ThR2_EH_pw00(Gw := Para.rT_ThR2_EH_Lim00, Hy := rT_ThR2_EH_PwLevHy, In := TK_moduleTR);
		xGRMax_ThR2_EH_pw20(Gw := Para.rT_ThR2_EH_Lim20, Hy := rT_ThR2_EH_PwLevHy, In := TK_moduleTR);
		xGRMax_ThR2_EH_pw40(Gw := Para.rT_ThR2_EH_Lim40, Hy := rT_ThR2_EH_PwLevHy, In := TK_moduleTR);
		xGRMax_ThR2_EH_pw60(Gw := Para.rT_ThR2_EH_Lim60, Hy := rT_ThR2_EH_PwLevHy, In := TK_moduleTR);
		xGRMax_ThR2_EH_pw80(Gw := Para.rT_ThR2_EH_Lim80, Hy := rT_ThR2_EH_PwLevHy, In := TK_moduleTR);

		IF FG_HEIZG_moduleTR = FALSE OR xGRMax_ThR2_EH_pw00.Q THEN
			iThR2_EH_PwLev := 0;
		ELSIF FG_HEIZG_moduleTR AND NOT(xGRMax_ThR2_EH_pw00.Q) AND xGRMax_ThR2_EH_pw20.Q THEN
			iThR2_EH_PwLev := 1;
		ELSIF FG_HEIZG_moduleTR AND NOT(xGRMax_ThR2_EH_pw00.Q) AND NOT(xGRMax_ThR2_EH_pw20.Q) AND xGRMax_ThR2_EH_pw40.Q THEN
			iThR2_EH_PwLev := 2;
		ELSIF FG_HEIZG_moduleTR AND NOT(xGRMax_ThR2_EH_pw00.Q) AND NOT(xGRMax_ThR2_EH_pw20.Q) AND NOT(xGRMax_ThR2_EH_pw40.Q) AND xGRMax_ThR2_EH_pw60.Q THEN
			iThR2_EH_PwLev := 3;
		ELSIF FG_HEIZG_moduleTR AND NOT(xGRMax_ThR2_EH_pw00.Q) AND NOT(xGRMax_ThR2_EH_pw20.Q) AND NOT(xGRMax_ThR2_EH_pw40.Q) AND NOT(xGRMax_ThR2_EH_pw60.Q) AND xGRMax_ThR2_EH_pw80.Q THEN
			iThR2_EH_PwLev := 4;
		ELSIF FG_HEIZG_moduleTR AND NOT(xGRMax_ThR2_EH_pw00.Q) AND NOT(xGRMax_ThR2_EH_pw20.Q) AND NOT(xGRMax_ThR2_EH_pw40.Q) AND NOT(xGRMax_ThR2_EH_pw60.Q) AND NOT(xGRMax_ThR2_EH_pw80.Q) THEN
			iThR2_EH_PwLev := 5;
		ELSE
			iThR2_EH_PwLev := 0;
		END_IF;

		//time ramp for el.heating power level
		xRamp_ThR2_EH_PwLev.In := INT_TO_REAL(iThR2_EH_PwLev);
		xRamp_ThR2_EH_PwLev();
		iThR2_EH_PwLev_ramp := TRUNC(xRamp_ThR2_EH_PwLev.Out);
		OUT_TR.rP_ThR_EH := INT_TO_REAL(iThR2_EH_PwLev_ramp) / 5 * 1000; (* 5 el.heating power levels, 1000 HMI display scaling factor *)

		//monitoring of heating elements groups availability depending on max.temperature
		xTON_ThR2_EH_gr1_T_GoodQual(IN := IN_TR.tT_ThR2_EH_group1.GoodQual, PT := tiTON_ThR2_EH_gr_T_GoodQual);
		xTON_ThR2_EH_gr2_T_GoodQual(IN := IN_TR.tT_ThR2_EH_group2.GoodQual, PT := tiTON_ThR2_EH_gr_T_GoodQual);
		xTON_ThR2_EH_gr3_T_GoodQual(IN := IN_TR.tT_ThR2_EH_group3.GoodQual, PT := tiTON_ThR2_EH_gr_T_GoodQual);
		xTON_ThR2_EH_gr4_T_GoodQual(IN := IN_TR.tT_ThR2_EH_group4.GoodQual, PT := tiTON_ThR2_EH_gr_T_GoodQual);
		xTON_ThR2_EH_gr5_T_GoodQual(IN := IN_TR.tT_ThR2_EH_group5.GoodQual, PT := tiTON_ThR2_EH_gr_T_GoodQual);

		xGRMax_ThR2_EH_group1_T(Gw := rT_ThR2_EH_thres_GroupHi, Hy := rT_ThR2_EH_thres_GroupHi_Hy, In := IN_TR.tT_ThR2_EH_group1.Ai);
		bThR2_EH_gr1_T_blocked := xGRMax_ThR2_EH_group1_T.Q AND xTON_ThR2_EH_gr1_T_GoodQual.Q;
		bThR2_EH_groupT_Ok[1] := NOT bThR2_EH_gr1_T_blocked;
		xGRMax_ThR2_EH_group2_T(Gw := rT_ThR2_EH_thres_GroupHi, Hy := rT_ThR2_EH_thres_GroupHi_Hy, In := IN_TR.tT_ThR2_EH_group2.Ai);
		bThR2_EH_gr2_T_blocked := xGRMax_ThR2_EH_group2_T.Q AND xTON_ThR2_EH_gr2_T_GoodQual.Q;
		bThR2_EH_groupT_Ok[2] := NOT bThR2_EH_gr2_T_blocked;
		xGRMax_ThR2_EH_group3_T(Gw := rT_ThR2_EH_thres_GroupHi, Hy := rT_ThR2_EH_thres_GroupHi_Hy, In := IN_TR.tT_ThR2_EH_group3.Ai);
		bThR2_EH_gr3_T_blocked := xGRMax_ThR2_EH_group3_T.Q AND xTON_ThR2_EH_gr3_T_GoodQual.Q;
		bThR2_EH_groupT_Ok[3] := NOT bThR2_EH_gr3_T_blocked;
		xGRMax_ThR2_EH_group4_T(Gw := rT_ThR2_EH_thres_GroupHi, Hy := rT_ThR2_EH_thres_GroupHi_Hy, In := IN_TR.tT_ThR2_EH_group4.Ai);
		bThR2_EH_gr4_T_blocked := xGRMax_ThR2_EH_group4_T.Q AND xTON_ThR2_EH_gr4_T_GoodQual.Q;
		bThR2_EH_groupT_Ok[4] := NOT bThR2_EH_gr4_T_blocked;
		xGRMax_ThR2_EH_group5_T(Gw := rT_ThR2_EH_thres_GroupHi, Hy := rT_ThR2_EH_thres_GroupHi_Hy, In := IN_TR.tT_ThR2_EH_group5.Ai);
		bThR2_EH_gr5_T_blocked := xGRMax_ThR2_EH_group5_T.Q AND xTON_ThR2_EH_gr5_T_GoodQual.Q;
		bThR2_EH_groupT_Ok[5] := NOT bThR2_EH_gr5_T_blocked;

		//definition of heating elements groups order based on flap position
		IF RM_KL_END THEN //flap in one of the end-positions with request
			IF RM_KL_END_EIN THEN //end-position right: heating element energization order right to left
				iThR2_EH_groupFirst := 5;
				iThR2_EH_groupLast := 1;
				iThR2_EH_groupIndexIncr := -1;
			ELSIF RM_KL_END_AUS THEN //end-position left: heating element energization order left to right
				iThR2_EH_groupFirst := 1;
				iThR2_EH_groupLast := 5;
				iThR2_EH_groupIndexIncr := 1;
			END_IF

			//set of heating elements groups status based on power level
			iThR2_EH_PwLevCounter := 0;
			FOR iThR2_EH_groupIndex := iThR2_EH_groupFirst TO iThR2_EH_groupLast BY iThR2_EH_groupIndexIncr DO
				IF bThR2_EH_groupT_Ok[iThR2_EH_groupIndex] AND (iThR2_EH_PwLevCounter < iThR2_EH_PwLev_ramp) THEN
					bThR2_EH_group_On[iThR2_EH_groupIndex] := TRUE;
					iThR2_EH_PwLevCounter := iThR2_EH_PwLevCounter + 1;
				ELSE
					bThR2_EH_group_On[iThR2_EH_groupIndex] := FALSE;
				END_IF
			END_FOR
			OUT_TR.tThR2_EH_group1_Dem.Do := bThR2_EH_group_On[1];
			OUT_TR.tThR2_EH_group2_Dem.Do := bThR2_EH_group_On[2];
			OUT_TR.tThR2_EH_group3_Dem.Do := bThR2_EH_group_On[3];
			OUT_TR.tThR2_EH_group4_Dem.Do := bThR2_EH_group_On[4];
			OUT_TR.tThR2_EH_group5_Dem.Do := bThR2_EH_group_On[5];
		ELSE
			OUT_TR.tThR2_EH_group1_Dem.Do := OUT_TR.tThR2_EH_group2_Dem.Do := OUT_TR.tThR2_EH_group3_Dem.Do := OUT_TR.tThR2_EH_group4_Dem.Do := OUT_TR.tThR2_EH_group5_Dem.Do := FALSE;
		END_IF
	ELSE
		//reset ramp in IF block
		xRamp_ThR2_EH_PwLev.In := 0;
		xRamp_ThR2_EH_PwLev();
		//reset timers in IF block
		xTON_ThR2_EH_gr1_T_GoodQual(IN := FALSE, PT := tiTON_ThR2_EH_gr_T_GoodQual);
		xTON_ThR2_EH_gr2_T_GoodQual(IN := FALSE, PT := tiTON_ThR2_EH_gr_T_GoodQual);
		xTON_ThR2_EH_gr3_T_GoodQual(IN := FALSE, PT := tiTON_ThR2_EH_gr_T_GoodQual);
		xTON_ThR2_EH_gr4_T_GoodQual(IN := FALSE, PT := tiTON_ThR2_EH_gr_T_GoodQual);
		xTON_ThR2_EH_gr5_T_GoodQual(IN := FALSE, PT := tiTON_ThR2_EH_gr_T_GoodQual);
		//reset all output signals to heating elements ThR2
		OUT_TR.tThR2_EH_group1_Dem.Do := OUT_TR.tThR2_EH_group2_Dem.Do := OUT_TR.tThR2_EH_group3_Dem.Do := OUT_TR.tThR2_EH_group4_Dem.Do := OUT_TR.tThR2_EH_group5_Dem.Do := FALSE;
	END_IF
	bThR_elHeating := OUT_TR.rP_ThR_EH > 0;

	(* Temperature Limits [FB33] *)

	(*
		IF (rP_Act_Norm_Filt >= 75) THEN bQ0 := 1;
	    ELSIF (rP_Act_Norm_Filt < 70) THEN bQ0 := 0;
		END_IF

		xTON_P_75(IN := bQ0, PT := T#2s);
		AN_P_75 := xTON_P_75.Q;

	*)

	(*************** temperature threshold check for TRW07 - ThR ***************)
	xGRMax_TK11(Gw := TKx_y_HI_Gw, Hy := TKx_y_HI_Hy, In := IN_TR.tT_ThR_Chamber1_1.Ai);

	xTON_TK1_1(IN := xGRMax_TK11.Q, PT := ti_TKx_y_HI_PTHI);
	xTK1_1_HI.QH  := xTON_TK1_1.Q;

	(****************************************)
	xGRMax_TK12(Gw := TKx_y_HI_Gw, Hy := TKx_y_HI_Hy, In := IN_TR.tT_ThR_Chamber1_2.Ai);

	xTON_TK1_2(IN := xGRMax_TK12.Q, PT := ti_TKx_y_HI_PTHI);
	xTK1_2_HI.QH   := xTON_TK1_2.Q;

	(****************************************)
	xGRMax_TK21(Gw := TKx_y_HI_Gw, Hy := TKx_y_HI_Hy, In := IN_TR.tT_ThR_Chamber2_1.Ai);

	xTON_TK2_1(IN := xGRMax_TK21.Q, PT := ti_TKx_y_HI_PTHI);
	xTK2_1_HI.QH  := xTON_TK2_1.Q;

	(****************************************)
	xGRMax_TK22(Gw := TKx_y_HI_Gw, Hy := TKx_y_HI_Hy, In := IN_TR.tT_ThR_Chamber2_2.Ai);

	xTON_TK2_2(IN := xGRMax_TK22.Q, PT := ti_TKx_y_HI_PTHI);
	xTK2_2_HI.QH  := xTON_TK2_2.Q;

	(*************** chamber temperature difference check for TRW06 - ThR ***************)
	IF FG_KLUM AND NOT Para.bThR2_Ena THEN
		TK1_DIF := ABS(IN_TR.tT_ThR_Chamber1_1.Ai  - IN_TR.tT_ThR_Chamber1_2.Ai);
	ELSE
		TK1_DIF := 0;
	END_IF;

	xGRMax_TK1DIF(Gw := rT_ThR_ChamberDiff, Hy := rT_ThR_ChamberDiffHy, In := TK1_DIF);
	xTON_TK1_DIF(IN := xGRMax_TK1DIF.Q, PT := ti_ThR_ChamberDiff);

	xGRMax_TK1Diff_switch(Gw := rT_ThR_ChDiff_switch, Hy := rT_ThR_ChDiff_switchHy, In := TK1_DIF);
	xTON_TK1_Diff_switch(IN := xGRMax_TK1Diff_switch.Q, PT := Para.ti_ThR_Val_y1);

	xTK1_DIF_HI.QH := xTON_TK1_DIF.Q OR xTON_TK1_Diff_switch.Q;

	(****************************************)
	IF FG_KLUM AND NOT Para.bThR2_Ena THEN
		TK2_DIF := ABS(IN_TR.tT_ThR_Chamber2_1.Ai - IN_TR.tT_ThR_Chamber2_2.Ai);
	ELSE
		TK2_DIF := 0;
	END_IF;

	xGRMax_TK2DIF(Gw := rT_ThR_ChamberDiff, Hy := rT_ThR_ChamberDiffHy, In := TK2_DIF);
	xTON_TK2_DIF(IN := xGRMax_TK2DIF.Q, PT := ti_ThR_ChamberDiff);

	xGRMax_TK2Diff_switch(Gw := rT_ThR_ChDiff_switch, Hy := rT_ThR_ChDiff_switchHy, In := TK2_DIF);
	xTON_TK2_Diff_switch(IN := xGRMax_TK2Diff_switch.Q, PT := Para.ti_ThR_Val_y1);

	xTK2_DIF_HI.QH := xTON_TK2_DIF.Q OR xTON_TK2_Diff_switch.Q;

	(*************** electrical heating temperature threshold check - ThR ***************)
	xGRMax_TK75(Gw := Para.rT_ThR_EH_Lim75, Hy := rT_ThR_EH_Lim75Hy, In := TK_moduleTR);
	xTK_E75.QH     := xGRMax_TK75.Q;

	(****************************************)
	xGRMax_TK50(Gw := Para.rT_ThR_EH_Lim50, Hy := rT_ThR_EH_Lim50Hy, In := TK_moduleTR);
	xTK_E50.QH     := xGRMax_TK50.Q;

	(****************************************)
	xGRMax_TK25(Gw := Para.rT_ThR_EH_Lim25, Hy := rT_ThR_EH_Lim25Hy, In := TK_moduleTR);
	xTK_E25.QH     := xGRMax_TK25.Q;

	(****************************************)
	xGRMax_TK00(Gw := Para.rT_ThR_EH_Lim00, Hy := rT_ThR_EH_Lim00Hy, In := TK_moduleTR);
	xTK_E00.QH     := xGRMax_TK00.Q;

	(*************** aux.gas release temperature threshold check ***************)
	xGRMax_TKG(Gw := Para.rT_ThR_LimGas, Hy := Para.rT_ThR_LimGasHy, In := TK1_TK2_MIN);
	xTK_GAS.QH     := xGRMax_TKG.Q;

	(*************** operating temperature threshold check ***************)
	xGRMax_ThR_OperTemp(Gw := TK_w + rT_ThR_OperTemp_rel, Hy := rT_ThR_OperTempHy, In := TK_moduleTR);
	xTK_OPER.QH := xGRMax_ThR_OperTemp.Q;

	(********************************************************************)

	(* Klappenumschaltzeit [FB40] *)
	IF (Para.bThR_woGas AND set_PT_KL_Pinc) THEN	(* set the flap flap switching interval on load increase value *)
		PTON_KL_AUS := Para.ti_ThR_ValIntervalPInc; (* Seconds --> Milliseconds --> TIME *)
		PTON_KL_EIN := PTON_KL_AUS;
	ELSE
		d := REAL_TO_DINT(polyg_2hl (REAL_TO_INT(TK1_TK2_MAX), ADR(PT_KL)));	(* Seconds *)
		PTON_KL_AUS := DINT_TO_TIME (d * 1000);    	(* Seconds --> Milliseconds --> TIME *)
		PTON_KL_EIN := PTON_KL_AUS;
	END_IF;

	(* Ansteuerung Gasregelventil [FB66] *)

	IF OUT_TR.bThR_RelGas THEN	// control valve close command timer selection for stop of aux. gas system
		tiTP_NFRG_GASREG := T#180s;	//default timer
	END_IF
	IF (NOT OUT_TR.bThR_RelGas AND xRS_Thr_AuxGasStopT.Q1) THEN
		tiTP_NFRG_GASREG := tiTON_Thr_AuxGasStopT_reset;	//reduced timer
	END_IF

	xTP_NFRG_GASREG (IN := NOT OUT_TR.bThR_RelGas, PT := tiTP_NFRG_GASREG);
	xTP_BTRB (IN := IN_TR.tEng_Run.Do, PT := T#180s);

	IF xTP_NFRG_GASREG.Q THEN
		OUT_TR.tThR_CV_CDec.Do := TRUE;
		OUT_TR.tThR_CV_CInc.Do := FALSE;
	ELSIF xTP_BTRB.Q THEN
		OUT_TR.tThR_CV_CDec.Do := TRUE;
		OUT_TR.tThR_CV_CInc.Do := FALSE;
	ELSIF OUT_TR.bThR_RelGas THEN
		OUT_TR.tThR_CV_CDec.Do := bCtrl_ThR_CDec;
		OUT_TR.tThR_CV_CInc.Do := bCtrl_ThR_CInc;
	ELSE
		OUT_TR.tThR_CV_CDec.Do := FALSE;
		OUT_TR.tThR_CV_CInc.Do := FALSE;
	END_IF;

	(******************************************************************************)
	(******************************************************************************)

	(* IntegralElement *)

	FOR x := 0 TO 1 BY 1 DO

		(* output:               Out: units "In"
		   internal calculation: Out_internal: units "In" *100
		                         dOut: 0,1 units "In"/s = 0,01 units "In"/0,1s
		                                                = 0,01 units "In"/sample *)

		IF P_ramp[x].mode = 1 THEN
			P_ramp[x].dOut_plus  :=
				(P_ramp[x].Ki_plus  * (P_ramp[x].In - P_ramp[x].Out)) / P_ramp[x].In_ref;
			P_ramp[x].dOut_minus :=
				(P_ramp[x].Ki_minus * (P_ramp[x].Out - P_ramp[x].In)) / P_ramp[x].In_ref;
		ELSE
			P_ramp[x].dOut_plus  := P_ramp[x].Ki_plus;
			P_ramp[x].dOut_minus := P_ramp[x].Ki_minus;
		END_IF;

		IF P_ramp[x].dOut_plus  < 1 THEN
			P_ramp[x].dOut_plus  := 1;
		ELSIF P_ramp[x].dOut_plus  > P_ramp[x].dOut_max_p THEN
			P_ramp[x].dOut_plus  := P_ramp[x].dOut_max_p;
		END_IF;

		IF P_ramp[x].dOut_minus < 1 THEN
			P_ramp[x].dOut_minus := 1;
		ELSIF P_ramp[x].dOut_minus > P_ramp[x].dOut_max_m THEN
			P_ramp[x].dOut_minus  := P_ramp[x].dOut_max_m;
		END_IF;

		P_ramp[x].In_internal := P_ramp[x].In;
		P_ramp[x].In_internal := P_ramp[x].In_internal * 100;

		(* Out > In: decrease Out *)
		IF P_ramp[x].Out_internal > P_ramp[x].In_internal THEN
			P_ramp[x].Out_internal := P_ramp[x].Out_internal - P_ramp[x].dOut_minus;
			IF P_ramp[x].Out_internal < P_ramp[x].In_internal THEN
				P_ramp[x].Out_internal := P_ramp[x].In_internal;
			END_IF;

		(* Out < In: increase Out *)
		ELSIF P_ramp[x].Out_internal < P_ramp[x].In_internal THEN
			P_ramp[x].Out_internal := P_ramp[x].Out_internal + P_ramp[x].dOut_plus;
			IF P_ramp[x].Out_internal > P_ramp[x].In_internal THEN
				P_ramp[x].Out_internal := P_ramp[x].In_internal;
			END_IF;
		END_IF;

		(* LIMIT Out_min, Out_max [units "In"]: *)
		IF P_ramp[x].Out_min < 0 THEN
			P_ramp[x].Out_min := 0;
		ELSIF P_ramp[x].Out_min > 32767 THEN
			P_ramp[x].Out_min := 32767;
		END_IF;
		IF P_ramp[x].Out_max < P_ramp[x].Out_min THEN
			P_ramp[x].Out_max := P_ramp[x].Out_min;
		ELSIF P_ramp[x].Out_max > 32767 THEN
			P_ramp[x].Out_max := 32767;
		END_IF;

		(* LIMIT Out_internal [units "In" *100]: *)
		IF P_ramp[x].Out_internal < (P_ramp[x].Out_min * 100) THEN
			P_ramp[x].Out_internal := P_ramp[x].Out_min * 100;
		ELSIF P_ramp[x].Out_internal > (P_ramp[x].Out_max * 100) THEN
			P_ramp[x].Out_internal := P_ramp[x].Out_max * 100;
		END_IF;

		P_ramp[x].Out := INT_TO_REAL(i32_t_i16 (REAL_TO_DINT(P_ramp[x].Out_internal)/100));	(* [units "In"] *)

	END_FOR;

END_PROGRAM
```

#### reactorInit.st
```iecst
(*******************************************************************************
AGGR: thermal reactor  (init)

This code is confidential AND proprietary TO the INNIO Company.
It may NOT be used in any form, OR reproduced in any manner, without the express
written permission OF the INNIO Company.
Copyright, INNIO Company, 2022

- initialize values used in main thermal reactor task

Customized modifications: -
------------------------

History:
-------
V4.12.0 12-05-2022	Maran	Initialization of values for fixed temperature thresholds
V4.13.0 27-03-2023	Maran	included operating temperature init, updated init values for max. temp. difference for W3503
V4.14.0 27-11-2024	Maran	added var. initializations for el. heating system and auxiliary gas solenoid valve for ThR2

Instructions FOR use:
--------------------

Outstandings:
------------
*******************************************************************************)

PROGRAM _INIT

// Th.Reactor maximum temperature warning - hysteresis and delay
TKx_y_HI_Hy			:=  20.0;  (* 0,1°C *)
ti_TKx_y_HI_PTHI	:= T#2s;

// Th.Reactor maximum temperature difference between TK1/TK2 warning - threshold, hysteresis and delay
rT_ThR_ChamberDiff		:=  50.0;  (* 0,1°C; Standard: 50,0 °C *)
rT_ThR_ChamberDiffHy :=  10.0;  (* 0,1°C *)
ti_ThR_ChamberDiff		:= T#60s;
rT_ThR_ChDiff_switch :=  20.0;
rT_ThR_ChDiff_switchHy :=  1.0;

// Th.Reactor electrical heating system - hysteresis for parameter limits
rT_ThR_EH_Lim75Hy		:= 20.0;        (* 0,1°C *)
rT_ThR_EH_Lim50Hy		:= 20.0;        (* 0,1°C *)
rT_ThR_EH_Lim25Hy		:= 20.0;        (* 0,1°C *)
rT_ThR_EH_Lim00Hy		:= 20.0;        (* 0,1°C *)
rT_ThR2_EH_PwLevHy		:= 20.0;

// Th.Reactor electrical heating system ThR2 - element group temperature monitoring threshold and hysteresis
rT_ThR2_EH_thres_GroupHi		:= 800;
rT_ThR2_EH_thres_GroupHi_Hy		:= 20;
tiTON_ThR2_EH_gr_T_GoodQual		:= T#30s;	// timer for monitoring temperature good quality signal

// Th.Reactor electrical heating system ThR2 - ramp rate for heating power increase/decrease
xRamp_ThR2_EH_PwLev.enable 		:=	TRUE;
xRamp_ThR2_EH_PwLev.Rise		:=	0.0333;			// 0.033 "In"/s
xRamp_ThR2_EH_PwLev.Sink		:=	100.0;			// 100 "In"/s, immediate decrease
xRamp_ThR2_EH_PwLev.TC_Time		:=	100;			// cycle Time 100ms

// Th.Reactor operating temperature - margin from setpoint and hysteresis
rT_ThR_OperTemp_rel		:=  -5.0;
rT_ThR_OperTempHy		:=  10.0;

// Th.Reactor auxiliary gas stop due to sufficient temperature - minimum margin above setpoint and timers
rT_Thr_AuxGasStopT_rel			:= 3.0;
tiTON_Thr_AuxGasStopT_set		:= T#12m;
tiTON_Thr_AuxGasStopT_reset		:= T#10s;
tiTP_NFRG_GASREG				:= T#180s;
rPos_ThR_GasCV_AuxGasStop_max	:= 0.03;

// Th.Reactor auxiliary gas solenoid valve ThR2 - timer for closing valve before flap switching
tiThR2_AuxGasValve_Block	:= T#5s;

END_PROGRAM
```

#### reactor_Local.var
```iecst
VAR
	d : DINT;
	FG_KLUM : BOOL;
	KL_AUS_S : BOOL;
	KL_EIN_S : BOOL;
	MS_TK : BOOL;
	PTON_KL_AUS : TIME;
	PTON_KL_EIN : TIME;
	PTON_SPLU_AKT_AUS : TIME;
	PTON_SPLU_AKT_EIN : TIME;
	PT_KL : coordinate_5;
	P_ramp : ARRAY[0..1] OF IntegralElement;
	RM_KL_END : BOOL;
	RM_KL_MIT : BOOL;
	SEK_TAKT : BOOL;
	SPLU_AKT : BOOL;
	ST_RM_ST : BOOL;
	ST_R_ST : BOOL;
	ti_TKx_y_HI_PTHI : TIME;
	TK1_TK2_MAX : REAL;
	TK1_TK2_MIN : REAL;
	TK1_TK2_MIT : REAL;
	TKx_y_HI_Gw : REAL; (*Reactor temperature TK1/TK2 maximum [degC]*)
	TKx_y_HI_Hy : REAL; (*Reactor temperature TK1/TK2 maximum - hysteresis [degC]*)
	rT_ThR_EH_Lim75Hy : REAL; (*Th.Reactor electrical heating system - hysteresis for 75% heating power [degC]*)
	rT_ThR_EH_Lim50Hy : REAL; (*Th.Reactor electrical heating system - hysteresis for 50% heating power [degC]*)
	rT_ThR_EH_Lim25Hy : REAL; (*Th.Reactor electrical heating system - hysteresis for 25% heating power [degC]*)
	rT_ThR_EH_Lim00Hy : REAL; (*Th.Reactor electrical heating system - hysteresis for 0% heating power [degC]*)
	TK_w : REAL; (*Th.Reactor - temperature setpoint [degC]*)
	x : INT; (*	XT_Version_32x : BOOL; *)
	xCTD_HE_1 : CTD;
	xCTD_HE_2 : CTD;
	xCTD_HE_3 : CTD;
	xGRMax_TK00 : GR_MAXR;
	xGRMax_TK11 : GR_MAXR;
	xGRMax_TK12 : GR_MAXR;
	xGRMax_TK21 : GR_MAXR;
	xGRMax_TK22 : GR_MAXR;
	xGRMax_TK25 : GR_MAXR;
	xGRMax_TK50 : GR_MAXR;
	xGRMax_TK75 : GR_MAXR;
	xGRMax_TKG : GR_MAXR;
	xR_TRIG_KL_AUS : R_TRIG;
	xR_TRIG_KL_EIN : R_TRIG;
	xTK1_1_HI : ls_t;
	xTK1_2_HI : ls_t;
	xTK1_DIF_HI : ls_t;
	xTK2_1_HI : ls_t;
	xTK2_2_HI : ls_t;
	xTK2_DIF_HI : ls_t;
	xTK_E00 : ls_t;
	xTK_E25 : ls;
	xTK_E50 : ls;
	xTK_E75 : ls;
	xTK_GAS : ls_t;
	xTK_OPER : ls_t;
	xTOF_PS_LUFT : TOF;
	xTOF_W_INT : TOF; (*weekly SPLU interval *)
	xTON_AUFHEIZG_GAS : TON;
	xTON_AUFHEIZG_GES : TON;
	xTON_FG_TH : TON;
	xTON_KL_AUS : TON;
	xTON_KL_EIN : TON;
	xTON_reactor_01 : TON;
	xTON_reactor_02 : TON;
	xTON_SPLU_AKT_AUS : TON;
	xTON_SPLU_AKT_EIN : TON;
	xTON_SPLU_DEAKT : TON;
	xTON_ST_KLE : TON;
	xTON_ST_KLM : TON;
	xTON_W_ACT : TON; (*weekly SPLU active*)
	xTP_BTRB : TP;
	xTP_NFRG_GASREG : TP;
	xTRW01_TK : SR;
	y_HE : REAL;
	y_HE_ramp : UINT;
	TK1_DIF : REAL := 0.0; (*Thermal reactor chamber TK1 temperature difference*)
	TK2_DIF : REAL := 0.0; (*Thermal reactor chamber TK2 temperature difference*)
	ti_ThR_ChamberDiff : TIME; (*Thermal reactor chamber temperatuer difference time interval before warning*)
	rT_ThR_ChamberDiffHy : REAL; (*Thermal reactor temperature difference hysteresis [degC]*)
	rT_ThR_ChamberDiff : REAL; (*Thermal reactor temperature difference [degC]*)
	xTON_TK1_DIF : TON;	(*auxiliary variable for warning W3503 - Th.Reactor chamber max temperature difference*)
	xTON_TK2_DIF : TON;	(*auxiliary variable for warning W3503 - Th.Reactor chamber max temperature difference*)
	xGRMax_TK1DIF : GR_MAXR; (*auxiliary variable for warning W3503 - Th.Reactor chamber max temperature difference*)
	xGRMax_TK2DIF : GR_MAXR; (*auxiliary variable for warning W3503 - Th.Reactor chamber max temperature difference*)
	rT_ThR_ChDiff_switch : REAL; (*Thermal reactor max. temperature difference during one valve switch period [degC]*)
	rT_ThR_ChDiff_switchHy : REAL; (*Thermal reactor chamber max temperature difference hysteresis [degC]*)
	xTON_TK1_Diff_switch : TON;	(*auxiliary variable for warning W3503 - Th.Reactor chamber max temperature difference*)
	xTON_TK2_Diff_switch : TON;	(*auxiliary variable for warning W3503 - Th.Reactor chamber max temperature difference*)
	xGRMax_TK1Diff_switch : GR_MAXR; (*auxiliary variable for warning W3503 - Th.Reactor chamber max temperature difference*)
	xGRMax_TK2Diff_switch : GR_MAXR; (*auxiliary variable for warning W3503 - Th.Reactor chamber max temperature difference*)
	R_TRIG_KL_AUS_M : R_TRIG;
	R_TRIG_KL_EIN_M : R_TRIG;
	xTOF_S_EIN : TOF;
	xTON_FG_KL_M : TON;
	xTON_KL_AUS_M : TON;
	xTON_KL_EIN_M : TON;
	R_TRIG_KL_AUS : R_TRIG;
	R_TRIG_KL_EIN : R_TRIG;
	KL_AUS_M : BOOL;
	KL_EIN_M : BOOL;
	FG_KL_M : BOOL;
	xTP_EH11 : TP;	(*aux. time pulse for thermal reactor electrical heating group 1*)
	xTP_EH21 : TP;	(*aux. time pulse for thermal reactor electrical heating group 2*)
	xTP_EH31 : TP;	(*aux. time pulse for thermal reactor electrical heating group 3*)
	rThR_EH_pulse : REAL;	(*aux. var. for thermal reactor electrical heating*)
	tThR_EH_pulse : TIME;	(*aux. var. for thermal reactor electrical heating*)
	xGRMax_ThR_OperTemp : GR_MAXR;
	rT_ThR_OperTemp_rel : REAL; (*Th.Reactor operating temperature - temperature margin from setpoint [degC]*)
	rT_ThR_OperTempHy : REAL; (*Thermal reactor operating temperature hysteresis [degC]*)
	bThr_AuxGasStopT_Ena : BOOL;	(* Th.Reactor auxiliary gas stop due to sufficient temperature - enabling conditions *)
	xTON_Thr_AuxGasStopT_set : TON;	(* TON timer for Th.Reactor auxiliary gas stop due to sufficient temperature *)
	tiTON_Thr_AuxGasStopT_set : TIME; (* auxiliary timer variable *)
	rT_Thr_AuxGasStopT_rel : REAL; (* Th.Reactor auxiliary gas stop due to sufficient temperature - temperature margin above setpoint [degC]*)
	xTON_Thr_AuxGasStopT_reset : TON;	(* TON timer for Th.Reactor auxiliary gas stop due to sufficient temperature *)
	tiTON_Thr_AuxGasStopT_reset : TIME; (* auxiliary timer variable *)
	rPos_ThR_GasCV_AuxGasStop_max: REAL; (* Thermal reactor  auxiliary gas stop due to sufficient temperature - maximum CV position for temperature verification validity [%] *)
	xRS_Thr_AuxGasStopT: RS;	(* Th.Reactor auxiliary gas stop due to sufficient temperature *)
	tiTP_NFRG_GASREG : TIME;	(* Th.Reactor aux. gas - control valve close command timer for stop of aux. gas system *)
	xGRMax_ThR2_EH_pw00 : GR_MAXR; (*Th.Reactor electrical heating system - ThR2 - threshold check 0% power [degC]*)
	xGRMax_ThR2_EH_pw20 : GR_MAXR; (*Th.Reactor electrical heating system - ThR2 - threshold check 20% power [degC]*)
	xGRMax_ThR2_EH_pw40 : GR_MAXR; (*Th.Reactor electrical heating system - ThR2 - threshold check 40% power [degC]*)
	xGRMax_ThR2_EH_pw60 : GR_MAXR; (*Th.Reactor electrical heating system - ThR2 - threshold check 60% power [degC]*)
	xGRMax_ThR2_EH_pw80 : GR_MAXR; (*Th.Reactor electrical heating system - ThR2 - threshold check 80% power [degC]*)
	rT_ThR2_EH_PwLevHy : REAL; (*Th.Reactor electrical heating system - ThR2 - hysteresis for heating power [degC]*)
	iThR2_EH_PwLev : INT; (*Th.Reactor electrical heating system - ThR2 - heating power level *)
	xRamp_ThR2_EH_PwLev : RAMPE_R; (*Th.Reactor electrical heating system - ThR2 - auxiliary variable *)
	iThR2_EH_PwLev_ramp : INT; (*Th.Reactor electrical heating system - ThR2 - heating power level *)
	xTON_ThR2_EH_gr1_T_GoodQual : TON;	(* TON timer for Th.Reactor electrical heating system - ThR2 - heating element group 1 temperature good quality signal *)
	xTON_ThR2_EH_gr2_T_GoodQual : TON;	(* TON timer for Th.Reactor electrical heating system - ThR2 - heating element group 1 temperature good quality signal *)
	xTON_ThR2_EH_gr3_T_GoodQual : TON;	(* TON timer for Th.Reactor electrical heating system - ThR2 - heating element group 1 temperature good quality signal *)
	xTON_ThR2_EH_gr4_T_GoodQual : TON;	(* TON timer for Th.Reactor electrical heating system - ThR2 - heating element group 1 temperature good quality signal *)
	xTON_ThR2_EH_gr5_T_GoodQual : TON;	(* TON timer for Th.Reactor electrical heating system - ThR2 - heating element group 1 temperature good quality signal *)
	tiTON_ThR2_EH_gr_T_GoodQual : TIME;	(* auxiliary timer variable *)
	xGRMax_ThR2_EH_group1_T : GR_MAXR; (*Th.Reactor electrical heating system - ThR2 - threshold check heating element group 1 high temperature [degC]*)
	xGRMax_ThR2_EH_group2_T : GR_MAXR; (*Th.Reactor electrical heating system - ThR2 - threshold check heating element group 2 high temperature [degC]*)
	xGRMax_ThR2_EH_group3_T : GR_MAXR; (*Th.Reactor electrical heating system - ThR2 - threshold check heating element group 3 high temperature [degC]*)
	xGRMax_ThR2_EH_group4_T : GR_MAXR; (*Th.Reactor electrical heating system - ThR2 - threshold check heating element group 4 high temperature [degC]*)
	xGRMax_ThR2_EH_group5_T : GR_MAXR; (*Th.Reactor electrical heating system - ThR2 - threshold check heating element group 5 high temperature [degC]*)
	rT_ThR2_EH_thres_GroupHi : REAL; (*Th.Reactor electrical heating system - ThR2 - heating elements high temperature threshold [degC]*)
	rT_ThR2_EH_thres_GroupHi_Hy : REAL; (*Th.Reactor electrical heating system - ThR2 - hysteresis for heating elements high temperature [degC]*)
	bThR2_EH_groupT_Ok : ARRAY[0..5] OF BOOL; (*Th.Reactor electrical heating system - ThR2 - availability status of heating element groups*)
	iThR2_EH_groupFirst  : INT; (*Th.Reactor electrical heating system - ThR2 - index of first group based on flap position*)
	iThR2_EH_groupLast  : INT; (*Th.Reactor electrical heating system - ThR2 - index of last group based on flap position*)
	iThR2_EH_groupIndex  : INT; (*Th.Reactor electrical heating system - ThR2 - heating element group index*)
	iThR2_EH_groupIndexIncr  : INT; (*Th.Reactor electrical heating system - ThR2 - increment of heating element group index*)
	iThR2_EH_PwLevCounter  : INT; (*Th.Reactor electrical heating system - ThR2 - auxiliary counter*)
	bThR2_EH_group_On : ARRAY[0..5] OF BOOL; (*Th.Reactor electrical heating system - ThR2 - energization request for heating element groups*)
	iThr2_lastFlapEndPosIndex  : INT; (*Th.Reactor - ThR2 - last end-position reached by 4-way flap *)
	xSR_Thr2_AuxGasValve_Block: SR;	(* Th.Reactor auxiliary gas solenoid valve - ThR2 *)
	tiThR2_AuxGasValve_Block : TIME; (* Th.Reactor auxiliary gas solenoid valve - ThR2 - time for closing valve before flap switching *)
	xGRMax_ThR2_T_LeftChamber_Hi : GR_MAXR; (*Th.Reactor - ThR2 - threshold check left chamber high temperature [degC]*)
	xGRMax_ThR2_T_RightChamber_Hi : GR_MAXR; (*Th.Reactor - ThR2 - threshold check right chamber high temperature [degC]*)
	xTON_ThR2_T_LeftChamber_Hi : TON; (* Th.Reactor - ThR2 - TON delay for warning - left chamber high temperature *)
	xTON_ThR2_T_RightChamber_Hi : TON; (* Th.Reactor - ThR2 - TON delay for warning - right chamber high temperature *)
END_VAR
```

#### how_to_do_reactor.txt - how to do:settings for reactor
```
----------------------------------------------------------------------------------------------
how to do the settings of "reactor"
V3.20.0 21-12-2010  Thaler (Update --)
----------------------------------------------------------------------------------------------

Select the type of temperature compensation for the thermocouples by "Compensation_AI_TK":
    up to V2.5x.x: in ReactorVarV2xxx.var
    from V2.60.0 upwards: in task "settings"

0 = internal (= Default):
if the compensating cables for thermocouples are installed till the input card AT6402 !
--> Compensation_AI_TK: value = 0
--> AT6402 / Open I/O Configuration: Function model 'internal compensation temperature'

1 = external universal:
if the compensating cables for thermocouples end in the terminal box of the reactor !
--> Compensation_AI_TK: value = 1
--> AT6402 / Open I/O Configuration: Function model 'external compensation temperature'
--> Open I/O Mapping, connect AI_Tvgl if applicable
--> if AI_Tvgl is type Pt100 or signal 20 mA:
    parameter Exhaust\Thermal reactor\Adjustment of the reference junction temperature = 20°C

2 = external type Pt100, 20 mA:
if the compensating cables for thermocouples end in the terminal box of the reactor, and
if the reference junction temperature measuring (AI_Tvgl) is done by Pt100 or signal 20 mA !
--> Compensation_AI_TK: value = 2
--> AT6402 / Open I/O Configuration: Function model 'external compensation temperature'
--> Open I/O Mapping, connect AI_Tvgl

----------------------------------------------------------------------------------------------

Select the type of position switches for the 4-way-flap by "UM_E_NEU" in task "reac_set":

value = 0: --> 4 limit switch positions = old version, used till 04.03.2010
           assigned inputs: DI_E_EIN_A, DI_E_EIN_E, DI_E_AUS_A, DI_E_AUS_E.

VALUE = 1: --> 3 limit switch positions (5 switches) = Default
           assigned Inputs: DI_KL_EIN1, DI_KL_EIN2, DI_E_MITT, DI_KL_AUS1, DI_KL_AUS2.

----------------------------------------------------------------------------------------------

Parameters:
Import the file "EXPORT_REAKTOR$$$.PAR" into the parameter file for the engine:
    EXPORT_REAKTOR V2.3x bis V2.6x yyy.PAR, resp.
    EXPORT_REAKTOR ab V3.1x.PAR

After the test bench / Before commissioning set the parameter
"Engine data\Thermal reactor" = 1 (User for write = 45)

----------------------------------------------------------------------------------------------
----------------------------------------------------------------------------------------------

for the version "without gas injection" apply additionally:

Task “reac_set”
    sel_woGas := TRUE;
    (* --> check/choose Reserve Parameter No. plant specific ! *)

Parameters:
Import additionally the following file into the parameter file for the engine:
    EXPORT_woGas V2.0 bis V2.6.PAR, resp.
    EXPORT_woGas ab V3.1.PAR
    (* --> check/choose Reserve Parameter No. plant specific ! *)

    from XT V3.1x.x upwards:
    use "ParaText.mdb" for the text of the reserve parameters

----------------------------------------------------------------------------------------------
```

- ParaText.mdb - Thermoreactor (binary file, 544768 bytes)
#### ReactorVarV3200_MS.var - Local variables
```iecst
(********************************************************************
 * COPYRIGHT -- INNIO Company
 ********************************************************************
 * File: ReaktorVarV3200.var
 * Author: ThJ
 * Created: Nov 18, 2010
 * Modified: Jun 10, 2011
  ********************************************************************
 * Global variables for reactor V3.20.0_MS,  SPS_moduleTR VER.:  >= A_V2501 <= A_V32xx
 ********************************************************************)
VAR
	xTON_TK2_1 : TON;
	xTON_TK1_2 : TON;
	xTON_TK2_2 : TON;
	xTON_TK1_1 : TON;
END_VAR
```

### Program Logical/ThermalReactor/Ctr_TR_4 (IEC) - Electric heater controller

#### Ctr_TR_4Cyclic.st - Cyclic code
```iecst
(*******************************************************************************
Ctr_TR_4		Controller Heater

This code is confidential AND proprietary TO the INNIO Company.
It may NOT be used in any form, or reproduced in any manner,
without the express written permission OF the INNIO Company.
Copyright, INNIO Company, 2022

Customized modifications: -
------------------------

History:
-------
V04.00.00	04-04-2014  Ganguly 		converted to modular software
V04.03.00	25-09-2014  Denk 			adjust step controller for Thermal reactor
V04.07.00	28-05-2019	Hohensinner 	new interfaces for CU Module (AB Energy like projects and so on)
V04.11.00	28-01-2022	Perktold		included plant controller upgrade
V04.12.00	18-05-2022	Maran			removed unused impulse time selection for step controller
V04.14.00	27-11-2024	Maran			update for thermal reactor 2nd generation (ThR2): blocked gas heater controller if aux. gas solenoid valve is closed

Instructions FOR use:
--------------------

Outstandings: -
------------
*******************************************************************************)

PROGRAM _CYCLIC

	(* Parameter *)
	Para.tCtrTR_Heater.W_set;
	Para.tCtrTR_Heater.W_set2;
	Para.tCtrTR_Heater.W_min;
	Para.tCtrTR_Heater.W_max;
	Para.tCtrTR_Heater.dW_up;
	Para.tCtrTR_Heater.dW_down;
	Para.tCtrTR_Heater.deadband;
	Para.tCtrTR_Heater.Y_min;
	Para.tCtrTR_Heater.Y_max;
	Para.tCtrTR_Heater.dY_max;
	Para.tCtrTR_Heater.Y_block;
	Para.tCtrTR_Heater.invert;
	Para.tCtrTR_Heater.Kp;
	Para.tCtrTR_Heater.Tn;
	Para.tCtrTR_Heater.Tv;
	Para.tCtrTR_Heater.Kp_GainScheduling;
	Para.tCtrTR_Heater.Tn_GainScheduling;
	Para.tCtrTR_Heater.Tv_GainScheduling;
	Para.tCtrTR_Heater.t_min_pulse_down;
	Para.tCtrTR_Heater.t_min_pulse_up;
	Para.tCtrTR_Heater.t_period_down;
	Para.tCtrTR_Heater.t_period_up;

	(* Input variables *)
	tCtrTR_Heater_In 				:= VIS2MM.tCtrTR_Heater_In;		(* from vis *)

	(* Input from module *)
	tCtrTR_Heater_In.enable       	:= 	Para.bThR_Active
									   	AND Para.bCtrThR_Heater_Active
										AND OUT_TR.bThR_RelGas
										AND NOT bThr2_AuxGasValve_CtrlBlock
										AND IN_TR.tPB2MM.bParaSetupOk;
	tCtrTR_Heater_In.W_ext_Active 	:= FALSE;
	tCtrTR_Heater_In.W_ext		  	:= 0.0;
	tCtrTR_Heater_In.Y_set_Active 	:= FALSE;
	tCtrTR_Heater_In.Y_set		  	:= 0.0;
	tCtrTR_Heater_In.X				:= TK_moduleTR;
	tCtrTR_Heater_In.A				:= 0.0;
	tCtrTR_Heater_In.W_set2_Active	:= FALSE;		(*Input to define which internal setpoint will be used TRUE = use the 2nd set point | FALSE use the normal "1st" one*)
	tCtrTR_Heater_In.GainScheduling	:= 0.0;			(*Input for Gain Scheduling: 0.0 = use 100% of the Standard PID-Parameters | 1.0 = use 100% of the GainSched. PID Parameters | linear interpolation in between*)
	tCtrTR_Heater_In.Y_min_cust		:= -1.0;		(*"customized" Y-Min at the current moment (The existing Y-Min parameter is the global minimum. To have an effect Y_min_cust needs to be > the parameter | -1.0 = function not used*)
	tCtrTR_Heater_In.Y_max_cust		:= 1.0;			(*"customized" Y-Max at the current moment (The existing Y-Max parameter is the global maximum. To have an effect Y_max_cust needs to be < the parameter | 1.0 = function not used*)
	tCtrTR_Heater_In.Retrigger		:= FALSE;		(*a rising edge on this input signals the controller to retrigger - set W on X and force the Integrator to the current Y*)

	IF bThr2_AuxGasValve_CtrlBlock THEN
		tCtrTR_Heater_In.Y_set_Active 	:= TRUE;
		tCtrTR_Heater_In.Y_set		  	:= tCtrTR_Heater_Out.Y;
	END_IF

	(* Input from Visualization via OPC *)
	tCtrTR_Heater_In.Y_man_Active;
	tCtrTR_Heater_In.Y_man;
	tCtrTR_Heater_In.X_min;
	tCtrTR_Heater_In.X_max;
	tCtrTR_Heater_In.Tune_quality;
	tCtrTR_Heater_In.Tune_PI;
	tCtrTR_Heater_In.Tune_PID;
	tCtrTR_Heater_In.Tune_start;
	tCtrTR_Heater_In.Tune_stop;
	tCtrTR_Heater_In.Tune_takeover;

	xCtrTR_Heater();

	(* Output variables function block *)
	(* Output to module(s) *)
	OUT_TR.tCtrTR_Heater_Set.Ao 	:= tCtrTR_Heater_Out.Y;

	OUT_TR.tCtrTR_Heater_Out		:=	tCtrTR_Heater_Out;

	(* Output to Visualization via OPC *)
	MM2VIS.tCtrTR_Heater_Out 		:= tCtrTR_Heater_Out;
	VIS2MM.tCtrTR_Heater_In  		:= tCtrTR_Heater_In;

	MM2VIS.tCtrTR_Heater_Out.Active;
	MM2VIS.tCtrTR_Heater_Out.Y;
	MM2VIS.tCtrTR_Heater_Out.W;
	MM2VIS.tCtrTR_Heater_Out.e;
	MM2VIS.tCtrTR_Heater_Out.Kp_tune;
	MM2VIS.tCtrTR_Heater_Out.Tn_tune;
	MM2VIS.tCtrTR_Heater_Out.Tv_tune;
	MM2VIS.tCtrTR_Heater_Out.status;
	MM2VIS.tCtrTR_Heater_Out.Step_down;
	MM2VIS.tCtrTR_Heater_Out.Step_up;

	(***********************************************************************************)
	(* Adjust step controller for Thermal reactor *)
	(* old plc_ctr4 #433 - 447 *)
	REG4_STELL 	:= FALSE;
	REG4_POS 	:= FALSE;
	REG4_NEG	:= FALSE;

	IF tCtrTR_Heater_Out.Y > 0.0 THEN						(* increasing the output value *)
		REG4_STELL 	:= TRUE;
		REG4_POS 	:= TRUE;
	END_IF

	IF tCtrTR_Heater_Out.Y < 0 THEN							(* decreasing the output value *)
		REG4_STELL 	:= TRUE;
		REG4_NEG 	:= TRUE;
	END_IF

	Y_absolut := (ABS(tCtrTR_Heater_Out.Y));				(* absolute value of the output *)

	(* Period duration (standard 10s), old NW46 *)
	xTOF_FA_T_REG4_1(IN := REG4_STELL AND NOT xTOF_FA_T_REG4_1.Q, PT := REAL_TO_TIME(Para.tCtrTR_Heater.t_period_up));
	T_REG4_1 := xTOF_FA_T_REG4_1.Q;

	tiImpulseTime := T#1s;
	(* Regulating time and regulating impulse for Step up, Teilweise NW48, NW50 *)
	xTP_FA_T_REG4_2_PLUS(IN := T_REG4_1, PT := tiImpulseTime/2);	(* Step up time control signal divided by 2*)
	T_REG4_2_PLUS := xTP_FA_T_REG4_2_PLUS.Q;

	(* Regulating time and regulating impulse for Step down, Teilweise NW49, NW50 *)
	xTP_FA_T_REG4_2_MINUS(IN := T_REG4_1, PT := tiImpulseTime);
	T_REG4_2_MINUS := xTP_FA_T_REG4_2_MINUS.Q;

	(* Control command Step up, NW52 *)
	Step_up 	:= Para.bThR_Active AND T_REG4_1 AND T_REG4_2_PLUS AND REG4_STELL AND REG4_POS;

	(* Control command Step down, NW54 *)
	Step_down 	:= Para.bThR_Active AND T_REG4_1 AND T_REG4_2_MINUS AND REG4_STELL AND REG4_NEG;

	(*********************************************************)
	(* Set control signal only when Y is constant increasing *)
	IF (tCtrTR_Heater_Out.Y > CntUp_old OR (tCtrTR_Heater_Out.Y > 0.999 AND tCtrTR_Heater_Out.Y < 1.001)) AND NOT bThr2_AuxGasValve_CtrlBlock THEN
		bCtrl_ThR_CInc := Step_up;				(* INFO: for standard controller step output insert here: tCtrTR_Heater_Out.Step_up *)
	ELSE
		bCtrl_ThR_CInc := FALSE;
	END_IF;
	CntUp_old := tCtrTR_Heater_Out.Y;

	(* Set control signal only when Y is constant decreasing *)
	IF (tCtrTR_Heater_Out.Y < CntDown_old OR (tCtrTR_Heater_Out.Y < -0.999 AND tCtrTR_Heater_Out.Y > -1.001)) AND NOT bThr2_AuxGasValve_CtrlBlock THEN
		bCtrl_ThR_CDec := Step_down;			(* INFO: for standard controller step output insert here: tCtrTR_Heater_Out.Step_down *)
	ELSE
		bCtrl_ThR_CDec := FALSE;
	END_IF;
	CntDown_old := tCtrTR_Heater_Out.Y;

END_PROGRAM
```

#### Ctr_TR_4Init.st - Initialization code
```iecst
(********************************************************************
 * COPYRIGHT -- INNIO Company
 ********************************************************************
 * Program: Ctr_TR_4
 * File: Ctr_TR_4Init.st
 * Author: 105051626
 * Created: November 08, 2013
 ********************************************************************
 * Implementation of program Ctr_TR_4
 ********************************************************************)

PROGRAM _INIT

	tCtrTR_Heater_In.W_ext_Active := FALSE;	// Thermal Reactor Heater controller in programmed to used internal set point.
	                                     	// It uses X_Set (internal set points) inputs

	Para.tCtrTR_Heater.Y_block := 0.0;  	// Force output to 0,0 when controller disabled.

	tCtrTR_Heater_In.AlwaysUseYRamp		:= TRUE;	(*If TRUE the Y signal will always limit the change rate via the according parameter | if FALSE the Y signal will jump in case the controller is disabled (blocked or set)*)
	tCtrTR_Heater_In.KeepYManAtBlock	:= TRUE;	(*If TRUE the controller will keep the Y-man value constant in case the controller is disabled (blocked or set) | If FALSE the blocked or set value will override the Y-man value*)
	tCtrTR_Heater_In.Y_min_cust			:= -1.0;	(*"customized" Y-Min at the current moment (The existing Y-Min parameter is the global minimum. To have an effect Y_min_cust needs to be > the parameter | -1.0 = function not used*)
	tCtrTR_Heater_In.Y_max_cust			:=  1.0;	(*"customized" Y-Max at the current moment (The existing Y-Max parameter is the global maximum. To have an effect Y_max_cust needs to be < the parameter | 1.0 = function not used*)
	tCtrTR_Heater_In.StepperMode		:= TRUE;	(* TRUE = use PWM-Mode (standard mode until 4.10) | FALSE = use continuous servo drive *)

	xCtrTR_Heater.pParameter := ADR(Para.tCtrTR_Heater);
	xCtrTR_Heater.pInput     := ADR(tCtrTR_Heater_In);
	xCtrTR_Heater.pOutput    := ADR(tCtrTR_Heater_Out);

END_PROGRAM
```

#### Ctr_TR_4.var - Local variables
```iecst
(********************************************************************
 * COPYRIGHT -- INNIO Company
 ********************************************************************
 * Program: Ctr_TR_4
 * File: Ctr_TR_4.var
 * Author: 105051626
 * Created: November 08, 2013
 ********************************************************************
 * Local variables of program Ctr_TR_4
 ********************************************************************)
VAR
	CntUp_old : REAL;
	CntDown_old : REAL;
	REG4_POS : BOOL; (* Postiver Stellbefehl *)
	REG4_NEG : BOOL; (* Postiver Stellbefehl *)
	REG4_STELL : BOOL; (* Stellbefehl *)
	T_REG4_1 : BOOL; (* Periodenzeit *)
	Y_absolut : REAL;
	tiImpulseTime : TIME;
	xTOF_FA_T_REG4_1 : TOF;
	xTP_FA_T_REG4_2_PLUS : TP;
	xTP_FA_T_REG4_2_MINUS : TP;
	T_REG4_2_PLUS : BOOL;
	T_REG4_2_MINUS : BOOL;
	Step_up : BOOL;
	Step_down : BOOL;
END_VAR
```

### Program Logical/ThermalReactor/MsgTR (IEC) - Messages

#### MsgTRCyclic.st - Cyclic code
```iecst
(*******************************************************************************
Msg_TR	 			 alarms generation MM_thermal reactor

This code is confidential and proprietary to the INNIO Company.
It may not be used in any form, or reproduced in any manner,
without written permission of the INNIO Company.
Copyright, INNIO Company, 2020

Customized modifications: -
------------------------

History:
-------
V04.00.00.00	02-11-2011	denk/ganguly	new
V04.09.00.00	20-02-2020	Denk 			Thermalreactor failure added
V04.10.00.00	24.11.2020	lettenb.		2356,2357,2358 added
V04.13.00.00	28.11.2023	Maran			warnings 9374, 9375, 9376, 9377, 9381 added
V04.14.00.00	27.11.2024	Maran			warnings 9501, 9502, 9396, 9397, 9398, 9503, 9500 for ThR2 added
											 disabled warnings 3498 and 3503 with ThR2
				27.11.2024	Maran			warnings 9504, 9505 for ThR2 added

Instructions for use:
--------------------
1) declare alarm with function block "Alm"
	declare buffert alarm bit MM2VIS.bMsg<message number>

2) use template to create a new alarm,
   substitue 0000 by alarm number and make settings:

	xMsg0000.Enable		:=	TRUE;		enable/disable alarm
	xMsg0000.Set		:=	FALSE;		alarm set condition
	xMsg0000.PT			:=	T#0s;		alarm delay time
	xMsg0000.Prio		:=	1;			alarm priority: 1-3 = trip, 4 = warning
	xMsg0000.RiskClass	:=	3;			risk class for remote alarm reset
	xMsg0000.Reset		:=	FALSE;		FALSE: for all standard alarms	prio 1,2,3 and warnings prio 4
										TRUE : for autoreset alarms

	MM2VIS.bMsg0000			:=	xMsg0000.Q;	connect buffert alarm bit for VIS and control

3)  expand INIT

3)	include datapoint into OPC configuration for vis

Outstandings: -
------------

(*******************************************************************************)

PROGRAM _CYCLIC

	(* reset general trip *)
	OUT_TR.tTR2AB.bGnlTrip1		:=	FALSE;
	OUT_TR.tTR2AB.bGnlTrip2		:=	FALSE;
	OUT_TR.tTR2AB.bGnlTrip3		:=	FALSE;
	OUT_TR.tTR2AB.bGnlWarning	:=	FALSE;
	OUT_TR.tTR2AB.bTriptype1	:=	FALSE;
	OUT_TR.tTR2AB.bTriptype2	:=	FALSE;
	OUT_TR.tTR2AB.bTriptype3	:=	FALSE;

	(* A2356 Earth fault auxiliaries power supply thermal reactor panel *)
	IN_TR.tTR_AuxPS_GndFault.Di := IN_TR.tTR_AuxPS_GndFault.Di OR NOT IN_TR.tTR_AuxPS_GndFault.GoodQual;

	xMsg2356.Enable		:=	TRUE;
	xMsg2356.Set		:=	NOT IN_TR.tTR_AuxPS_GndFault.Di;
	xMsg2356.PT			:=	T#0s;
	xMsg2356.Prio		:=	2;
	xMsg2356.RiskClass	:=	4;
	xMsg2356.Reset		:=	FALSE;
	xMsg2356();
	MM2VIS.bMsg2356		:=	xMsg2356.Q;

	(* A2357 Auxiliaries power supply circuit breaker thermal reactor panel tripped *)
	IN_TR.tTR_AuxPS_CB_Trip.Di := IN_TR.tTR_AuxPS_CB_Trip.Di OR NOT IN_TR.tTR_AuxPS_CB_Trip.GoodQual;

	xMsg2357.Enable		:=	TRUE;
	xMsg2357.Set		:=	NOT IN_TR.tTR_AuxPS_CB_Trip.Di;
	xMsg2357.PT			:=	T#0s;
	xMsg2357.Prio		:=	2;
	xMsg2357.RiskClass	:=	4;
	xMsg2357.Reset		:=	FALSE;
	xMsg2357();
	MM2VIS.bMsg2357		:=	xMsg2357.Q;

	(* A2358 Auxiliaries power supply circuit breaker thermal reactor panel opened *)
	IN_TR.tTR_AuxPS_CB_On.Di := IN_TR.tTR_AuxPS_CB_On.Di OR NOT IN_TR.tTR_AuxPS_CB_On.GoodQual;

	xMsg2358.Enable		:=	TRUE;
	xMsg2358.Set		:=	NOT IN_TR.tTR_AuxPS_CB_On.Di;
	xMsg2358.PT			:=	T#0s;
	xMsg2358.Prio		:=	2;
	xMsg2358.RiskClass	:=	4;
	xMsg2358.Reset		:=	FALSE;
	xMsg2358();
	MM2VIS.bMsg2358		:=	xMsg2358.Q;

	(* bMsg 3306 Alarm - Disturbance exhaust valve middle position *)
	xMsg3306.Enable		:=	Para.bThR_Active;
	xMsg3306.Set		:=	xTRA01.Q1;
	xMsg3306.PT			:=	T#0s;
	xMsg3306.Prio		:=	2;
	xMsg3306.RiskClass	:=	4;
	xMsg3306.Reset		:=	FALSE;
	xMsg3306();
	MM2VIS.bMsg3306		:=	xMsg3306.Q;

	(* bMsg 3307 Alarm - Safety loop thermal reactor, active only with RIO *)
	xMsg3307.Enable		:=	Para.bThR_Active;
	xMsg3307.Set		:=	xTRA02.Q1;
	xMsg3307.PT			:=	T#0s;
	xMsg3307.Prio		:=	2;
	xMsg3307.RiskClass	:=	4;
	xMsg3307.Reset		:=	FALSE;
	xMsg3307();
	MM2VIS.bMsg3307		:=	xMsg3307.Q;

	(* bMsg 3498 Warning - Sensor failure *)
	xMsg3498.Enable		:=	Para.bThR_Active AND NOT Para.bThR2_Ena;
	xMsg3498.Set		:=	xTRW01.Q1;
	xMsg3498.PT			:=	T#0s;
	xMsg3498.Prio		:=	4;
	xMsg3498.RiskClass	:=	4;
	xMsg3498.Reset		:=	FALSE;
	xMsg3498();
	MM2VIS.bMsg3498		:=	xMsg3498.Q;

	(* bMsg 9501 Warning - Measuring signal failure thermal reactor temperature right side - ThR2 *)
	xMsg9501.Enable		:=	Para.bThR_Active AND Para.bThR2_Ena AND IN_TR.tPB2MM.bParaSetupOk;
	xMsg9501.Set		:=	NOT IN_TR.tThR2_T_UnitOk_RightCh.Di OR NOT IN_TR.tT_ThR2_RightChamber.GoodQual;
	xMsg9501.PT			:=	T#0s;
	xMsg9501.Prio		:=	4;
	xMsg9501.RiskClass	:=	4;
	xMsg9501.Reset		:=	FALSE;
	xMsg9501();
	MM2VIS.bMsg9501		:=	xMsg9501.Q;

	(* bMsg 9502 Warning - Measuring signal failure thermal reactor temperature left side - ThR2 *)
	xMsg9502.Enable		:=	Para.bThR_Active AND Para.bThR2_Ena AND IN_TR.tPB2MM.bParaSetupOk;
	xMsg9502.Set		:=	NOT IN_TR.tThR2_T_UnitOk_LeftCh.Di OR NOT IN_TR.tT_ThR2_LeftChamber.GoodQual;
	xMsg9502.PT			:=	T#0s;
	xMsg9502.Prio		:=	4;
	xMsg9502.RiskClass	:=	4;
	xMsg9502.Reset		:=	FALSE;
	xMsg9502();
	MM2VIS.bMsg9502		:=	xMsg9502.Q;

	(* bMsg 3499 Warning - Disturbance in pressurized air supply *)
	xMsg3499.Enable		:=	Para.bThR_Active;
	xMsg3499.Set		:=	xTRW02.Q1;
	xMsg3499.PT			:=	T#0s;
	xMsg3499.Prio		:=	4;
	xMsg3499.RiskClass	:=	4;
	xMsg3499.Reset		:=	FALSE;
	xMsg3499();
	MM2VIS.bMsg3499		:=	xMsg3499.Q;

	(* bMsg 3500 Warning - Disturbance in exhaust valve end position *)
	xMsg3500.Enable		:=	Para.bThR_Active;
	xMsg3500.Set		:=	xTRW03.Q1;
	xMsg3500.PT			:=	T#0s;
	xMsg3500.Prio		:=	4;
	xMsg3500.RiskClass	:=	4;
	xMsg3500.Reset		:=	FALSE;
	xMsg3500();
	MM2VIS.bMsg3500		:=	xMsg3500.Q;

	(* bMsg 3501 Warning - Heating time exceeded *)
	xMsg3501.Enable		:=	Para.bThR_Active;
	xMsg3501.Set		:=	xTRW04.Q1;
	xMsg3501.PT			:=	T#0s;
	xMsg3501.Prio		:=	4;
	xMsg3501.RiskClass	:=	4;
	xMsg3501.Reset		:=	FALSE;
	xMsg3501();
	MM2VIS.bMsg3501		:=	xMsg3501.Q;

	(* bMsg 3502 Warning - Control panel temperature too high *)
	xMsg3502.Enable		:=	Para.bThR_Active;
	xMsg3502.Set		:=	xTRW05.Q1;
	xMsg3502.PT			:=	T#0s;
	xMsg3502.Prio		:=	4;
	xMsg3502.RiskClass	:=	4;
	xMsg3502.Reset		:=	FALSE;
	xMsg3502();
	MM2VIS.bMsg3502		:=	xMsg3502.Q;

	(* bMsg 3503 Warning - Temperature difference between TK1/TK2 over allowed maximum *)
	xMsg3503.Enable		:=	Para.bThR_Active AND NOT Para.bThR2_Ena;
	xMsg3503.Set		:=	xTRW06.Q1;
	xMsg3503.PT			:=	T#0s;
	xMsg3503.Prio		:=	4;
	xMsg3503.RiskClass	:=	4;
	xMsg3503.Reset		:=	FALSE;
	xMsg3503();
	MM2VIS.bMsg3503		:=	xMsg3503.Q;

	(* bMsg 3504 Warning - Reactor temperature TK1/TK2 maximum *)
	xMsg3504.Enable		:=	Para.bThR_Active;
	xMsg3504.Set		:=	xTRW07.Q1;
	xMsg3504.PT			:=	T#0s;
	xMsg3504.Prio		:=	4;
	xMsg3504.RiskClass	:=	4;
	xMsg3504.Reset		:=	FALSE;
	xMsg3504();
	MM2VIS.bMsg3504		:=	xMsg3504.Q;

	(* bMsg 3505 Warning - Reactor temperature minimum *)
	xMsg3505.Enable		:=	Para.bThR_Active;
	xMsg3505.Set		:=	xTRW08.Q1;
	xMsg3505.PT			:=	T#0s;
	xMsg3505.Prio		:=	4;
	xMsg3505.RiskClass	:=	4;
	xMsg3505.Reset		:=	FALSE;
	xMsg3505();
	MM2VIS.bMsg3505		:=	xMsg3505.Q;

	(* bMsg 9374 Warning - Measuring signal failure auxiliary gas control valve position *)
	xMsg9374.Enable		:=	Para.bThR_Active AND Para.bThR_auxGasMonitor AND IN_TR.tPB2MM.bParaSetupOk;
	xMsg9374.Set		:=	NOT IN_TR.tPos_ThR_AuxGasCV_Act.GoodQual;
	xMsg9374.PT			:=	T#0s;
	xMsg9374.Prio		:=	4;
	xMsg9374.RiskClass	:=	4;
	xMsg9374.Reset		:=	FALSE;
	xMsg9374();
	MM2VIS.bMsg9374		:=	xMsg9374.Q;

	(* bMsg 9375 Warning - Measuring signal failure auxiliary gas pressure before control valve *)
	xMsg9375.Enable		:=	Para.bThR_Active AND Para.bThR_auxGasMonitor AND IN_TR.tPB2MM.bParaSetupOk;
	xMsg9375.Set		:=	NOT IN_TR.tPr_ThR_AuxGasBeforeCV.GoodQual;
	xMsg9375.PT			:=	T#0s;
	xMsg9375.Prio		:=	4;
	xMsg9375.RiskClass	:=	4;
	xMsg9375.Reset		:=	FALSE;
	xMsg9375();
	MM2VIS.bMsg9375		:=	xMsg9375.Q;

	(* bMsg 9376 Warning - Measuring signal failure auxiliary gas pressure after control valve *)
	xMsg9376.Enable		:=	Para.bThR_Active AND Para.bThR_auxGasMonitor AND IN_TR.tPB2MM.bParaSetupOk;
	xMsg9376.Set		:=	NOT IN_TR.tPr_ThR_AuxGasAfterCV.GoodQual;
	xMsg9376.PT			:=	T#0s;
	xMsg9376.Prio		:=	4;
	xMsg9376.RiskClass	:=	4;
	xMsg9376.Reset		:=	FALSE;
	xMsg9376();
	MM2VIS.bMsg9376		:=	xMsg9376.Q;

	(* bMsg 9377 Warning - Thermal reactor auxiliary gas compressor fault, low pressure before control valve *)
	xMsg9377.Enable		:=	Para.bThR_Active AND Para.bThR_auxGasMonitor;
	xMsg9377.Set		:=	bThr_AuxGasCompressor_Fault;
	xMsg9377.PT			:=	T#0s;
	xMsg9377.Prio		:=	4;
	xMsg9377.RiskClass	:=	4;
	xMsg9377.Reset		:=	FALSE;
	xMsg9377();
	MM2VIS.bMsg9377		:=	xMsg9377.Q;

	(* bMsg 9381 Warning - Thermal reactor implausible auxiliary gas pressure before/after control valve *)
	xMsg9381.Enable		:=	Para.bThR_Active AND Para.bThR_auxGasMonitor;
	xMsg9381.Set		:=	bThr_AuxGasPr_PcheckFail;
	xMsg9381.PT			:=	T#0s;
	xMsg9381.Prio		:=	4;
	xMsg9381.RiskClass	:=	4;
	xMsg9381.Reset		:=	FALSE;
	xMsg9381();
	MM2VIS.bMsg9381		:=	xMsg9381.Q;

	(* bMsg 9396 Warning - Thermal reactor: differential pressure maximum - ThR2 *)
	xMsg9396.Enable		:=	Para.bThR_Active AND IN_TR.tPB2MM.bParaSetupOk;
	xMsg9396.Set		:=	bThR2_DPr_Hi;
	xMsg9396.PT			:=	T#0s;
	xMsg9396.Prio		:=	4;
	xMsg9396.RiskClass	:=	4;
	xMsg9396.Reset		:=	FALSE;
	xMsg9396();
	MM2VIS.bMsg9396		:=	xMsg9396.Q;

	(* bMsg 9397 Warning - Measuring signal failure thermal reactor inlet pressure - ThR2 *)
	xMsg9397.Enable		:=	Para.bThR_Active AND Para.bThR2_Ena AND IN_TR.tPB2MM.bParaSetupOk;
	xMsg9397.Set		:=	NOT IN_TR.tPr_ThR2_Inlet.GoodQual;
	xMsg9397.PT			:=	T#0s;
	xMsg9397.Prio		:=	4;
	xMsg9397.RiskClass	:=	4;
	xMsg9397.Reset		:=	FALSE;
	xMsg9397();
	MM2VIS.bMsg9397		:=	xMsg9397.Q;

	(* bMsg 9398 Warning - Measuring signal failure thermal reactor outlet pressure - ThR2 *)
	xMsg9398.Enable		:=	Para.bThR_Active AND Para.bThR2_Ena AND IN_TR.tPB2MM.bParaSetupOk;
	xMsg9398.Set		:=	NOT IN_TR.tPr_ThR2_Outlet.GoodQual;
	xMsg9398.PT			:=	T#0s;
	xMsg9398.Prio		:=	4;
	xMsg9398.RiskClass	:=	4;
	xMsg9398.Reset		:=	FALSE;
	xMsg9398();
	MM2VIS.bMsg9398		:=	xMsg9398.Q;

	(* bMsg 9503 Warning - Measuring signal failure thermal reactor downstream temperature - ThR2 *)
	xMsg9503.Enable		:=	Para.bThR_Active AND Para.bThR2_Ena AND IN_TR.tPB2MM.bParaSetupOk;
	xMsg9503.Set		:=	NOT IN_TR.tThR2_T_UnitOk_Downstream.Di OR NOT IN_TR.tT_ThR2_Downstream.GoodQual;
	xMsg9503.PT			:=	T#0s;
	xMsg9503.Prio		:=	4;
	xMsg9503.RiskClass	:=	4;
	xMsg9503.Reset		:=	FALSE;
	xMsg9503();
	MM2VIS.bMsg9503		:=	xMsg9503.Q;

	(* bMsg 9500 Warning - Measuring signal failure electrical heating monitoring temperature sensors - ThR2 *)
	xMsg9500.Enable		:=	Para.bThR_Active AND Para.bThR2_Ena AND IN_TR.tPB2MM.bParaSetupOk;
	xMsg9500.Set		:=	NOT IN_TR.tT_ThR2_EH_group1.GoodQual OR NOT IN_TR.tT_ThR2_EH_group2.GoodQual OR NOT IN_TR.tT_ThR2_EH_group3.GoodQual OR NOT IN_TR.tT_ThR2_EH_group4.GoodQual OR NOT IN_TR.tT_ThR2_EH_group5.GoodQual;
	xMsg9500.PT			:=	T#0s;
	xMsg9500.Prio		:=	4;
	xMsg9500.RiskClass	:=	4;
	xMsg9500.Reset		:=	FALSE;
	xMsg9500();
	MM2VIS.bMsg9500		:=	xMsg9500.Q;

	(* bMsg 9504 Warning - Thermal reactor auxiliary gas injection solenoid valve fault - ThR2 *)
	xMsg9504.Enable		:=	Para.bThR_Active AND Para.bThR2_Ena;
	xMsg9504.Set		:=	bThr2_AuxGasValve_fault;
	xMsg9504.PT			:=	T#0s;
	xMsg9504.Prio		:=	4;
	xMsg9504.RiskClass	:=	4;
	xMsg9504.Reset		:=	FALSE;
	xMsg9504();
	MM2VIS.bMsg9504		:=	xMsg9504.Q;

	(* bMsg 9505 Warning - Exhaust aftertreatment: Thermal reactor outlet/SCR inlet high differential pressure - ThR2 *)
	xMsg9505.Enable		:=	Para.bThR_Active AND Para.bThR2_Ena AND (Para.bSCR_Active OR Para.bSCR_Cust_Active) AND IN_TR.tPB2MM.bParaSetupOk;
	xMsg9505.Set		:=	bThR2out_SCRin_DPr_Hi;
	xMsg9505.PT			:=	T#0s;
	xMsg9505.Prio		:=	4;
	xMsg9505.RiskClass	:=	4;
	xMsg9505.Reset		:=	FALSE;
	xMsg9505();
	MM2VIS.bMsg9505		:=	xMsg9505.Q;

	(* bMsg 9309  Warning - Thermo reactor failure / not in operation *)
	xMsg9309.Enable		:=	TRUE;
	xMsg9309.Set		:=	bThR_Failure;
	xMsg9309.PT			:=	T#0s;
	xMsg9309.Prio		:=	4;
	xMsg9309.RiskClass	:=	4;
	xMsg9309.Reset		:=	FALSE;
	xMsg9309();
	MM2VIS.bMsg9309		:=	xMsg9309.Q;

	(* B9042 Thermal reactor: operating switch OFF *)
	xMsg9042.Enable		:=	TRUE;
	xMsg9042.Set		:=	OUT_TR.bThR_Active AND NOT IN_TR.tThR_Swth_On.Di;
	xMsg9042.Reset		:=	TRUE;
	xMsg9042();
	MM2VIS.bMsg9042		:=	xMsg9042.Q;

	(* B9043 Thermal reactor: operating switch ON *)
	xMsg9043.Enable		:=	TRUE;
	xMsg9043.Set		:=	OUT_TR.bThR_Active AND IN_TR.tThR_Swth_On.Di;
	xMsg9043.Reset		:=	TRUE;
	xMsg9043();
	MM2VIS.bMsg9043		:=	xMsg9043.Q;

	(*--------------------------------------------------------------------------*)
	(* general alarms for further module operations *)
	bGnlTrip1	:= OUT_TR.tTR2AB.bGnlTrip1   OR IN_TR.tAB2TR.bGnlTrip1;
	bGnlTrip2	:= OUT_TR.tTR2AB.bGnlTrip2   OR IN_TR.tAB2TR.bGnlTrip2;
	bGnlTrip3	:= OUT_TR.tTR2AB.bGnlTrip3   OR IN_TR.tAB2TR.bGnlTrip3;
	bGnlWarning	:= OUT_TR.tTR2AB.bGnlWarning OR IN_TR.tAB2TR.bGnlWarning;

	bGnlTrip	:=	bGnlTrip1 OR bGnlTrip2 OR bGnlTrip3;

	(*******************************************************************************)
END_PROGRAM
```

#### MsgTRInit.st - Initialization code
```iecst
(*******************************************************************************
Msg_TR	 			 alarms generation MM_Thermal Reactor

This code is confidential and proprietary to the INNIO Company.
It may not be used in any form, or reproduced in any manner,
without written permission of the INNIO Company.
Copyright, INNIO Company, 2020

Customized modifications: -
------------------------

History:
-------
V0.00.0	01.11.2013	denk/ganguly	new

Instructions for use:
--------------------
1) declare alarm with function block "Msg"

2) use template to create a new alarm, substitue 0000 by message number:

	xMsg0000.Num		:=	0000;					alarm number
	xMsg0000.AmmInAdr	:=  iAdrAmmBase2MM;			do not change
	xMsg0000.AmmOutAdr	:=  iAdrMM2AmmBase;			do not change

3) 	set alarm number

Outstandings:
------------
(*******************************************************************************)
PROGRAM _INIT

	iAdrAmmBase2MM		:=  ADR(IN_TR.tAB2TR);
	iAdrMM2AmmBase		:=  ADR(OUT_TR.tTR2AB);

	(*******************************************************************************)

	xMsg2356.Num		:=	2356;
	xMsg2356.AmmInAdr	:=  iAdrAmmBase2MM;
	xMsg2356.AmmOutAdr	:=  iAdrMM2AmmBase;

	xMsg2357.Num		:=	2357;
	xMsg2357.AmmInAdr	:=  iAdrAmmBase2MM;
	xMsg2357.AmmOutAdr	:=  iAdrMM2AmmBase;

	xMsg2358.Num		:=	2358;
	xMsg2358.AmmInAdr	:=  iAdrAmmBase2MM;
	xMsg2358.AmmOutAdr	:=  iAdrMM2AmmBase;

	xMsg3306.Num		:=	3306;
	xMsg3306.AmmInAdr	:=  iAdrAmmBase2MM;
	xMsg3306.AmmOutAdr	:=  iAdrMM2AmmBase;

	xMsg3307.Num		:=	3307;
	xMsg3307.AmmInAdr	:=  iAdrAmmBase2MM;
	xMsg3307.AmmOutAdr	:=  iAdrMM2AmmBase;

	xMsg3498.Num		:=	3498;
	xMsg3498.AmmInAdr	:=  iAdrAmmBase2MM;
	xMsg3498.AmmOutAdr	:=  iAdrMM2AmmBase;

	xMsg9501.Num		:=	9501;
	xMsg9501.AmmInAdr	:=  iAdrAmmBase2MM;
	xMsg9501.AmmOutAdr	:=  iAdrMM2AmmBase;

	xMsg9502.Num		:=	9502;
	xMsg9502.AmmInAdr	:=  iAdrAmmBase2MM;
	xMsg9502.AmmOutAdr	:=  iAdrMM2AmmBase;

	xMsg3499.Num		:=	3499;
	xMsg3499.AmmInAdr	:=  iAdrAmmBase2MM;
	xMsg3499.AmmOutAdr	:=  iAdrMM2AmmBase;

	xMsg3500.Num		:=	3500;
	xMsg3500.AmmInAdr	:=  iAdrAmmBase2MM;
	xMsg3500.AmmOutAdr	:=  iAdrMM2AmmBase;

	xMsg3501.Num		:=	3501;
	xMsg3501.AmmInAdr	:=  iAdrAmmBase2MM;
	xMsg3501.AmmOutAdr	:=  iAdrMM2AmmBase;

	xMsg3502.Num		:=	3502;
	xMsg3502.AmmInAdr	:=  iAdrAmmBase2MM;
	xMsg3502.AmmOutAdr	:=  iAdrMM2AmmBase;

	xMsg3503.Num		:=	3503;
	xMsg3503.AmmInAdr	:=  iAdrAmmBase2MM;
	xMsg3503.AmmOutAdr	:=  iAdrMM2AmmBase;

	xMsg3504.Num		:=	3504;
	xMsg3504.AmmInAdr	:=  iAdrAmmBase2MM;
	xMsg3504.AmmOutAdr	:=  iAdrMM2AmmBase;

	xMsg3505.Num		:=	3505;
	xMsg3505.AmmInAdr	:=  iAdrAmmBase2MM;
	xMsg3505.AmmOutAdr	:=  iAdrMM2AmmBase;

	xMsg9374.Num		:=	9374;
	xMsg9374.AmmInAdr	:=  iAdrAmmBase2MM;
	xMsg9374.AmmOutAdr	:=  iAdrMM2AmmBase;

	xMsg9375.Num		:=	9375;
	xMsg9375.AmmInAdr	:=  iAdrAmmBase2MM;
	xMsg9375.AmmOutAdr	:=  iAdrMM2AmmBase;

	xMsg9376.Num		:=	9376;
	xMsg9376.AmmInAdr	:=  iAdrAmmBase2MM;
	xMsg9376.AmmOutAdr	:=  iAdrMM2AmmBase;

	xMsg9377.Num		:=	9377;
	xMsg9377.AmmInAdr	:=  iAdrAmmBase2MM;
	xMsg9377.AmmOutAdr	:=  iAdrMM2AmmBase;

	xMsg9381.Num		:=	9381;
	xMsg9381.AmmInAdr	:=  iAdrAmmBase2MM;
	xMsg9381.AmmOutAdr	:=  iAdrMM2AmmBase;

	xMsg9396.Num		:=	9396;
	xMsg9396.AmmInAdr	:=  iAdrAmmBase2MM;
	xMsg9396.AmmOutAdr	:=  iAdrMM2AmmBase;

	xMsg9397.Num		:=	9397;
	xMsg9397.AmmInAdr	:=  iAdrAmmBase2MM;
	xMsg9397.AmmOutAdr	:=  iAdrMM2AmmBase;

	xMsg9398.Num		:=	9398;
	xMsg9398.AmmInAdr	:=  iAdrAmmBase2MM;
	xMsg9398.AmmOutAdr	:=  iAdrMM2AmmBase;

	xMsg9503.Num		:=	9503;
	xMsg9503.AmmInAdr	:=  iAdrAmmBase2MM;
	xMsg9503.AmmOutAdr	:=  iAdrMM2AmmBase;

	xMsg9500.Num		:=	9500;
	xMsg9500.AmmInAdr	:=  iAdrAmmBase2MM;
	xMsg9500.AmmOutAdr	:=  iAdrMM2AmmBase;

	xMsg9504.Num		:=	9504;
	xMsg9504.AmmInAdr	:=  iAdrAmmBase2MM;
	xMsg9504.AmmOutAdr	:=  iAdrMM2AmmBase;

	xMsg9505.Num		:=	9505;
	xMsg9505.AmmInAdr	:=  iAdrAmmBase2MM;
	xMsg9505.AmmOutAdr	:=  iAdrMM2AmmBase;

	xMsg9309.Num		:=  9309;
	xMsg9309.AmmInAdr	:=  iAdrAmmBase2MM;
	xMsg9309.AmmOutAdr	:=  iAdrMM2AmmBase;

	xMsg9042.Num		:=  9042;
	xMsg9042.AmmInAdr	:=  iAdrAmmBase2MM;
	xMsg9042.AmmOutAdr	:=  iAdrMM2AmmBase;

	xMsg9043.Num		:=  9043;
	xMsg9043.AmmInAdr	:=  iAdrAmmBase2MM;
	xMsg9043.AmmOutAdr	:=  iAdrMM2AmmBase;

END_PROGRAM
```

#### MsgTR.var - Local variables
```iecst
(********************************************************************
 * COPYRIGHT -- INNIO Company
 ********************************************************************
 * Program: MsgTR
 * File: MsgTR.var
 * Author: 105051626
 * Created: November 01, 2013
 ********************************************************************
 * Local variables of program MsgTR
 ********************************************************************)
VAR
	iAdrMM2AmmBase : UDINT;
	iAdrAmmBase2MM : UDINT;
	xMsg2356 : Msg;
	xMsg2357 : Msg;
	xMsg2358 : Msg;
	xMsg3306 : Msg;
	xMsg3307 : Msg;
	xMsg3498 : Msg;
	xMsg9501 : Msg;
	xMsg9502 : Msg;
	xMsg3499 : Msg;
	xMsg3500 : Msg;
	xMsg3501 : Msg;
	xMsg3502 : Msg;
	xMsg3503 : Msg;
	xMsg3504 : Msg;
	xMsg3505 : Msg;
	xMsg9374 : Msg;
	xMsg9375 : Msg;
	xMsg9376 : Msg;
	xMsg9377 : Msg;
	xMsg9381 : Msg;
	xMsg9396 : Msg;
	xMsg9397 : Msg;
	xMsg9398 : Msg;
	xMsg9503 : Msg;
	xMsg9500 : Msg;
	xMsg9504 : Msg;
	xMsg9505 : Msg;
	xMsg9309 : Msg;
	xMsg9042 : Msg;
	xMsg9043 : Msg;
END_VAR
```

### Program Logical/ThermalReactor/ParTR (IEC) - + Parameter handling

- perm_par.st (not readable text: treated as protected, skipped)

#### perm_par.var
```iecst
VAR
	tParaIntern : ParaHandler_typ; (*Connector type to perm_par*)
	tMM2ParaBase_ReadBack : MM2ParaBase_type; (*INTERNAL! V4.06 new readback structure for information from previous tasks*)
	bWriteDataObj : BOOL; (* TRUE=write data object module *)
	bDataObjLenErr : BOOL; (*Error occured in permem: data module size missmatch*)
	bCreateDataObj : BOOL; (* TRUE=create new data object *)
	bWriteOnce : BOOL; (* write permanent memory once *)
	DatObjCreate_01 : DatObjCreate; (* data object create *)
	DatObjInfoBak_02 : DatObjInfo; (* data object info *)
	DatObjDelete_01 : DatObjDelete; (* data object delete *)
	DatObjRead_01 : DatObjRead; (* data object read *)
	DatObjRead_02 : DatObjRead; (* manual initiated data object read *)
	DatObjWrite_01 : DatObjWrite; (* data object write *)
	DatObjDelete_02 : DatObjDelete; (* data object delete *)
	DatObjDelete_11 : DatObjDelete; (*Delete Backup File*)
	DatObjInfo_01 : DatObjInfo; (* data object info *)
	DatObjInfo_02 : DatObjInfo; (* data object info *)
	szModuleName : STRING[35]; (* module name of object *)
	szModuleNameBackup : STRING[35]; (* module name of posiibly created backup object *)
	DatObjCopy_01 : DatObjCopy;
	bCopyDataObj : BOOL;
	TON_WarnDelay : TON;
	TON_WritePMEM : TON; (* delay write permanent memory *)
	ulPMPointer : UDINT; (* adress of actual checksum value *)
	ulChecksum : UDINT; (* parameter checksum value *)
	pm_len : UDINT; (* permanent value lenght *)
	ulChecksumOld : UDINT; (* last vlaue of parameter checksum *)
	ulChkValue : UDINT; (* actual value of parameter pointer *)
	pm_id : UDINT; (* permanent value identifier *)
	pm_p : UDINT; (* permanent value pointer *)
	DatObjInfo_META : DatObjInfo;
	DatObjRead_META : DatObjRead;
	szMetaDataRaw : STRING[2000];
	szMetaData : ARRAY[0..4] OF STRING[35];
	szMetaDataVis : ARRAY[0..3] OF STRING[35];
	ssIndex : INT;
	ssCount : INT;
	ucMetaDataRaw : ARRAY[0..2000] OF USINT;
	ssCount2 : INT;
	szMetaDataFile : STRING[10];
	szText1 : STRING[20];
	pv_adr_IN_XX_tPB2MM : UDINT;
	pv_lng : UDINT;
	pv_lng_IN_XX_tPB2MM : UDINT;
	pv_lng_OUT_XX_tPB2MM : UDINT;
	szText2 : STRING[20];
	pv_adr_OUT_XX_tXX2PB : UDINT;
END_VAR
VAR CONSTANT
	ERR_NOERROR : UINT := 0;
END_VAR
VAR
	usPMWriteCnt : UINT;
	pm_Error : UDINT; (* permanent value error *) (* Deleted: pm : ParaMem_typ; permanent memory tags mathias, 22.8.11*)
	fun_Error : UDINT := 0; (*state > 0 = function error*)
	xLocalParaCheck : ParaCheckFUB; (*local function instance to check parameter values*)
	TON_ParaSetupOk : TON;
	bParaCheckSystemOk : BOOL;
	iDebug_ParaOkChecked : UDINT;
	bRestoreBackupDataObj : BOOL := FALSE;
	bRestoreDataObjContent : BOOL := FALSE;
	pm_id_backup : UDINT;
	pm_p_Backup : UDINT;
	DatObjCopy_02 : DatObjCopy;
	bDeleteBackupDataObj : BOOL := FALSE; (*Command to delete backup data module file on purpose*)
	bDebugPara : ARRAY[0..5] OF BOOL;
	ssIndex2 : INT;
	ssIndex3 : INT;
	ssIndex4 : INT;
	ssIndexVis : INT;
	szText : STRING[40];
	pv_adr_Para : UDINT;
	szParaSnippet : ARRAY[0..5] OF STRING[150];
	szParaIndex : STRING[10];
	slValue : DINT;
	iModuleDLD_ResetCount : INT;
	bDownloadDetected : BOOL;
	bFlagParaStructCopyWorking : BOOL; (*true, if cyclic para copying is active, 1 false cycle at every copy *)
	bStoreInitParaInDataObj : BOOL := FALSE;
	bTestflag : BOOL;
	bReadOutMETA_Once : BOOL;
	tParaCheck_iPvAdress : ARRAY[0..5] OF UDINT;
	tParaCheck_iPvLengt : ARRAY[0..5] OF UDINT;
	tParaCheck_rPvValue : ARRAY[0..5] OF REAL;
	tParaCheck_rRangeMIN : ARRAY[0..5] OF REAL;
	tParaCheck_rRangeMAX : ARRAY[0..5] OF REAL;
	tParaCheck_szPvName : ARRAY[0..5] OF STRING[35];
	ssFormatDetected : INT;
	szMetaDataPart : STRING[150];
	szFullTaskName : STRING[35];
	szFullMetaModuleName : STRING[35];
	debugLen : INT;
	debugSize : INT := 0;
	strcat_adr1 : UDINT;
	strcat_adr2 : UDINT;
	ssIndexTN : INT;
	bAlternate : BOOL;
	n : INT;
	iAlternateChecksum : DINT;
	iAlternateChecksumOld : DINT;
	ulDebugChkValue : ARRAY[0..999] OF UDINT;
	Adr1 : UDINT;
	Adr2 : UDINT;
	usPMWriteCntStepsize : UINT := 1; (*different step sizes to help debug*)
	usPMWriteCntXOR : UINT;
	usPMWriteCntAltSum : UINT;
	ulAdrPM : UDINT;
	usChkValuePM : USINT;
	ulAdrPara : UDINT;
	ulPara_len : UDINT;
	usChkValuePara : USINT;
	iDebugCountPMDifferences : DINT := 0;
	bEngineRunDetected : BOOL; (*detection status bit autocommand 100 /101  for engine run state*)
	ucMetaDataDebugInfoLine : ARRAY[0..24] OF STRING[80];
	ssIndexMand : INT := 0;
	szMetaDataMand : STRING[35];
	iMyErrorInfo_Autoreset : DINT; (*internal autoreset counter*)
	ssIndex_Version : INT; (*internal*)
	ssIndex_BU : INT; (*internal*)
	ssIndex_BU2 : INT; (*internal*)
END_VAR
```

### Program Logical/ThermalReactor/PermTR (IEC) - + Permanent stored data

- perm_par.st (not readable text: treated as protected, skipped)
